KUKA KRL data list: CNC5.dat

&ACCESS RV
DEFDAT CNC5 Public
DECL GLOBAL FRAME gfCNCPoint5[30000]


gfCNCPoint5[1] = {X 169.9145, Y 15.4818, Z -6.3333, A 0.000, B 0.000, C 0.000 }
gfCNCPoint5[2] = {X 169.6699, Y 14.6462, Z -6.3333, A 0.000, B 0.000, C 0.000 }
gfCNCPoint5[3] = {X 169.6011, Y 13.7783, Z -6.3333, A 0.000, B 0.000, C 0.000 }
gfCNCPoint5[4] = {X 169.7111, Y 12.9146, Z -6.3333, A 0.000, B 0.000, C 0.000 }
gfCNCPoint5[5] = {X 169.9952, Y 12.0915, Z -6.3333, A 0.000, B 0.000, C 0.000 }
gfCNCPoint5[6] = {X 170.4414, Y 11.3439, Z -6.3333, A 0.000, B 0.000, C 0.000 }
gfCNCPoint5[7] = {X 171.0309, Y 10.7031, Z -6.3333, A 0.000, B 0.000, C 0.000 }
gfCNCPoint5[8] = {X 171.7389, Y 10.1963, Z -6.3333, A 0.000, B 0.000, C 0.000 }
gfCNCPoint5[9] = {X 172.3689, Y 9.8371, Z -6.3333, A 0.000, B 0.000, C 0.000 }
gfCNCPoint5[10] = {X 173.2226, Y 9.4761, Z -6.3333, A 0.000, B 0.000, C 0.000 }
gfCNCPoint5[11] = {X 174.1343, Y 9.3093, Z -6.3333, A 0.000, B 0.000, C 0.000 }
gfCNCPoint5[12] = {X 175.0605, Y 9.3446, Z -6.3333, A 0.000, B 0.000, C 0.000 }
gfCNCPoint5[13] = {X 175.9569, Y 9.5802, Z -6.3333, A 0.000, B 0.000, C 0.000 }
gfCNCPoint5[14] = {X 177.1785, Y 9.1095, Z -6.3333, A 0.000, B 0.000, C 0.000 }
gfCNCPoint5[15] = {X 179.3486, Y 8.3113, Z -6.3333, A 0.000, B 0.000, C 0.000 }
gfCNCPoint5[16] = {X 181.5872, Y 7.7326, Z -6.3333, A 0.000, B 0.000, C 0.000 }
gfCNCPoint5[17] = {X 183.8722, Y 7.3791, Z -6.3333, A 0.000, B 0.000, C 0.000 }
gfCNCPoint5[18] = {X 186.1811, Y 7.2543, Z -6.3333, A 0.000, B 0.000, C 0.000 }
gfCNCPoint5[19] = {X 188.4909, Y 7.3595, Z -6.3333, A 0.000, B 0.000, C 0.000 }
gfCNCPoint5[20] = {X 190.7789, Y 7.6937, Z -6.3333, A 0.000, B 0.000, C 0.000 }
gfCNCPoint5[21] = {X 192.7312, Y 8.2006, Z -6.3333, A 0.000, B 0.000, C 0.000 }
gfCNCPoint5[22] = {X 194.6099, Y 8.9351, Z -6.3333, A 0.000, B 0.000, C 0.000 }
gfCNCPoint5[23] = {X 196.3884, Y 9.8866, Z -6.3333, A 0.000, B 0.000, C 0.000 }
gfCNCPoint5[24] = {X 198.0419, Y 11.0420, Z -6.3333, A 0.000, B 0.000, C 0.000 }
gfCNCPoint5[25] = {X 199.0952, Y 11.9790, Z -6.3333, A 0.000, B 0.000, C 0.000 }
gfCNCPoint5[26] = {X 200.0403, Y 13.0251, Z -6.3333, A 0.000, B 0.000, C 0.000 }
gfCNCPoint5[27] = {X 200.8660, Y 14.1678, Z -6.3333, A 0.000, B 0.000, C 0.000 }
gfCNCPoint5[28] = {X 201.5625, Y 15.3935, Z -6.3333, A 0.000, B 0.000, C 0.000 }
gfCNCPoint5[29] = {X 202.1217, Y 16.6876, Z -6.3333, A 0.000, B 0.000, C 0.000 }
gfCNCPoint5[30] = {X 202.5931, Y 18.3350, Z -6.3333, A 0.000, B 0.000, C 0.000 }
gfCNCPoint5[31] = {X 202.8729, Y 20.0254, Z -6.3333, A 0.000, B 0.000, C 0.000 }
gfCNCPoint5[32] = {X 202.9574, Y 21.7368, Z -6.3333, A 0.000, B 0.000, C 0.000 }
gfCNCPoint5[33] = {X 202.8453, Y 23.4466, Z -6.3333, A 0.000, B 0.000, C 0.000 }
gfCNCPoint5[34] = {X 202.5383, Y 25.1324, Z -6.3333, A 0.000, B 0.000, C 0.000 }
gfCNCPoint5[35] = {X 202.0887, Y 26.5970, Z -6.3333, A 0.000, B 0.000, C 0.000 }
gfCNCPoint5[36] = {X 201.4503, Y 27.9897, Z -6.3333, A 0.000, B 0.000, C 0.000 }
gfCNCPoint5[37] = {X 200.6341, Y 29.2863, Z -6.3333, A 0.000, B 0.000, C 0.000 }
gfCNCPoint5[38] = {X 199.6544, Y 30.4641, Z -6.3333, A 0.000, B 0.000, C 0.000 }
gfCNCPoint5[39] = {X 198.5281, Y 31.5028, Z -6.3333, A 0.000, B 0.000, C 0.000 }
gfCNCPoint5[40] = {X 199.3593, Y 31.8268, Z -6.3333, A 0.000, B 0.000, C 0.000 }
gfCNCPoint5[41] = {X 200.1043, Y 32.3175, Z -6.3333, A 0.000, B 0.000, C 0.000 }
gfCNCPoint5[42] = {X 200.7302, Y 32.9532, Z -6.3333, A 0.000, B 0.000, C 0.000 }
gfCNCPoint5[43] = {X 201.2091, Y 33.7058, Z -6.3333, A 0.000, B 0.000, C 0.000 }
gfCNCPoint5[44] = {X 204.2502, Y 39.9879, Z -6.3333, A 0.000, B 0.000, C 0.000 }
gfCNCPoint5[45] = {X 204.5648, Y 40.8802, Z -6.3333, A 0.000, B 0.000, C 0.000 }
gfCNCPoint5[46] = {X 204.6737, Y 41.8200, Z -6.3333, A 0.000, B 0.000, C 0.000 }
gfCNCPoint5[47] = {X 204.5715, Y 42.7606, Z -6.3333, A 0.000, B 0.000, C 0.000 }
gfCNCPoint5[48] = {X 204.2633, Y 43.6551, Z -6.3333, A 0.000, B 0.000, C 0.000 }
gfCNCPoint5[49] = {X 203.7643, Y 44.4590, Z -6.3333, A 0.000, B 0.000, C 0.000 }
gfCNCPoint5[50] = {X 203.0996, Y 45.1323, Z -6.3333, A 0.000, B 0.000, C 0.000 }
gfCNCPoint5[51] = {X 202.5635, Y 45.5657, Z -6.3333, A 0.000, B 0.000, C 0.000 }
gfCNCPoint5[52] = {X 201.8660, Y 46.0245, Z -6.3333, A 0.000, B 0.000, C 0.000 }
gfCNCPoint5[53] = {X 201.0922, Y 46.3381, Z -6.3333, A 0.000, B 0.000, C 0.000 }
gfCNCPoint5[54] = {X 200.2721, Y 46.4943, Z -6.3333, A 0.000, B 0.000, C 0.000 }
gfCNCPoint5[55] = {X 199.4373, Y 46.4873, Z -6.3333, A 0.000, B 0.000, C 0.000 }
gfCNCPoint5[56] = {X 198.6199, Y 46.3171, Z -6.3333, A 0.000, B 0.000, C 0.000 }
gfCNCPoint5[57] = {X 196.5061, Y 47.4225, Z -6.3333, A 0.000, B 0.000, C 0.000 }
gfCNCPoint5[58] = {X 194.3068, Y 48.3461, Z -6.3333, A 0.000, B 0.000, C 0.000 }
gfCNCPoint5[59] = {X 192.0377, Y 49.0815, Z -6.3333, A 0.000, B 0.000, C 0.000 }
gfCNCPoint5[60] = {X 189.8324, Y 49.5923, Z -6.3333, A 0.000, B 0.000, C 0.000 }
gfCNCPoint5[61] = {X 187.5867, Y 49.8772, Z -6.3333, A 0.000, B 0.000, C 0.000 }
gfCNCPoint5[62] = {X 185.3237, Y 49.9332, Z -6.3333, A 0.000, B 0.000, C 0.000 }
gfCNCPoint5[63] = {X 183.0667, Y 49.7599, Z -6.3333, A 0.000, B 0.000, C 0.000 }
gfCNCPoint5[64] = {X 180.8388, Y 49.3589, Z -6.3333, A 0.000, B 0.000, C 0.000 }
gfCNCPoint5[65] = {X 179.0075, Y 48.8281, Z -6.3333, A 0.000, B 0.000, C 0.000 }
gfCNCPoint5[66] = {X 177.2496, Y 48.0897, Z -6.3333, A 0.000, B 0.000, C 0.000 }
gfCNCPoint5[67] = {X 175.5885, Y 47.1536, Z -6.3333, A 0.000, B 0.000, C 0.000 }
gfCNCPoint5[68] = {X 174.0464, Y 46.0322, Z -6.3333, A 0.000, B 0.000, C 0.000 }
gfCNCPoint5[69] = {X 172.9127, Y 44.9979, Z -6.3333, A 0.000, B 0.000, C 0.000 }
gfCNCPoint5[70] = {X 171.9093, Y 43.8366, Z -6.3333, A 0.000, B 0.000, C 0.000 }
gfCNCPoint5[71] = {X 171.0504, Y 42.5648, Z -6.3333, A 0.000, B 0.000, C 0.000 }
gfCNCPoint5[72] = {X 170.3480, Y 41.2003, Z -6.3333, A 0.000, B 0.000, C 0.000 }
gfCNCPoint5[73] = {X 169.8121, Y 39.7622, Z -6.3333, A 0.000, B 0.000, C 0.000 }
gfCNCPoint5[74] = {X 169.4500, Y 38.2708, Z -6.3333, A 0.000, B 0.000, C 0.000 }
gfCNCPoint5[75] = {X 169.3946, Y 37.9230, Z -6.3333, A 0.000, B 0.000, C 0.000 }
gfCNCPoint5[76] = {X 165.4444, Y 38.5519, Z -6.3333, A 0.000, B 0.000, C 0.000 }
gfCNCPoint5[77] = {X 165.4444, Y 38.5520, Z -6.3333, A 0.000, B 0.000, C 0.000 }
gfCNCPoint5[78] = {X 169.4737, Y 37.9104, Z -6.3333, A 0.000, B 0.000, C 0.000 }
gfCNCPoint5[79] = {X 169.4183, Y 37.5626, Z -6.3333, A 0.000, B 0.000, C 0.000 }
gfCNCPoint5[80] = {X 169.2618, Y 35.9753, Z -6.3333, A 0.000, B 0.000, C 0.000 }
gfCNCPoint5[81] = {X 169.2787, Y 34.3803, Z -6.3333, A 0.000, B 0.000, C 0.000 }
gfCNCPoint5[82] = {X 169.4688, Y 32.7966, Z -6.3333, A 0.000, B 0.000, C 0.000 }
gfCNCPoint5[83] = {X 169.8298, Y 31.2430, Z -6.3333, A 0.000, B 0.000, C 0.000 }
gfCNCPoint5[84] = {X 170.3575, Y 29.7378, Z -6.3333, A 0.000, B 0.000, C 0.000 }
gfCNCPoint5[85] = {X 171.0238, Y 28.3859, Z -6.3333, A 0.000, B 0.000, C 0.000 }
gfCNCPoint5[86] = {X 171.8736, Y 27.1412, Z -6.3333, A 0.000, B 0.000, C 0.000 }
gfCNCPoint5[87] = {X 172.8900, Y 26.0283, Z -6.3333, A 0.000, B 0.000, C 0.000 }
gfCNCPoint5[88] = {X 174.0526, Y 25.0692, Z -6.3333, A 0.000, B 0.000, C 0.000 }
gfCNCPoint5[89] = {X 175.3386, Y 24.2832, Z -6.3333, A 0.000, B 0.000, C 0.000 }
gfCNCPoint5[90] = {X 174.4745, Y 23.9351, Z -6.3333, A 0.000, B 0.000, C 0.000 }
gfCNCPoint5[91] = {X 173.7095, Y 23.4034, Z -6.3333, A 0.000, B 0.000, C 0.000 }
gfCNCPoint5[92] = {X 173.0820, Y 22.7148, Z -6.3333, A 0.000, B 0.000, C 0.000 }
gfCNCPoint5[93] = {X 172.6235, Y 21.9039, Z -6.3333, A 0.000, B 0.000, C 0.000 }
gfCNCPoint5[94] = {X 169.9886, Y 15.4516, Z -6.3333, A 0.000, B 0.000, C 0.000 }
gfCNCPoint5[95] = {X 169.7252, Y 14.4911, Z -6.3333, A 0.000, B 0.000, C 0.000 }
gfCNCPoint5[96] = {X 169.6977, Y 13.4955, Z -6.3333, A 0.000, B 0.000, C 0.000 }
gfCNCPoint5[97] = {X 169.9076, Y 12.5218, Z -6.3333, A 0.000, B 0.000, C 0.000 }
gfCNCPoint5[98] = {X 170.3429, Y 11.6260, Z -6.3333, A 0.000, B 0.000, C 0.000 }
gfCNCPoint5[99] = {X 170.9787, Y 10.8594, Z -6.3333, A 0.000, B 0.000, C 0.000 }
gfCNCPoint5[100] = {X 171.7785, Y 10.2658, Z -6.3333, A 0.000, B 0.000, C 0.000 }
gfCNCPoint5[101] = {X 172.4082, Y 9.9068, Z -6.3333, A 0.000, B 0.000, C 0.000 }
gfCNCPoint5[102] = {X 173.2457, Y 9.5527, Z -6.3333, A 0.000, B 0.000, C 0.000 }
gfCNCPoint5[103] = {X 174.1402, Y 9.3891, Z -6.3333, A 0.000, B 0.000, C 0.000 }
gfCNCPoint5[104] = {X 175.0488, Y 9.4237, Z -6.3333, A 0.000, B 0.000, C 0.000 }
gfCNCPoint5[105] = {X 175.9283, Y 9.6549, Z -6.3333, A 0.000, B 0.000, C 0.000 }
gfCNCPoint5[106] = {X 176.0174, Y 9.6904, Z -6.3333, A 0.000, B 0.000, C 0.000 }
gfCNCPoint5[107] = {X 177.2098, Y 9.1831, Z -6.3333, A 0.000, B 0.000, C 0.000 }
gfCNCPoint5[108] = {X 179.3724, Y 8.3877, Z -6.3333, A 0.000, B 0.000, C 0.000 }
gfCNCPoint5[109] = {X 181.6033, Y 7.8109, Z -6.3333, A 0.000, B 0.000, C 0.000 }
gfCNCPoint5[110] = {X 183.8805, Y 7.4587, Z -6.3333, A 0.000, B 0.000, C 0.000 }
gfCNCPoint5[111] = {X 186.1814, Y 7.3343, Z -6.3333, A 0.000, B 0.000, C 0.000 }
gfCNCPoint5[112] = {X 188.4833, Y 7.4392, Z -6.3333, A 0.000, B 0.000, C 0.000 }
gfCNCPoint5[113] = {X 190.7634, Y 7.7722, Z -6.3333, A 0.000, B 0.000, C 0.000 }
gfCNCPoint5[114] = {X 192.7066, Y 8.2767, Z -6.3333, A 0.000, B 0.000, C 0.000 }
gfCNCPoint5[115] = {X 194.5764, Y 9.0077, Z -6.3333, A 0.000, B 0.000, C 0.000 }
gfCNCPoint5[116] = {X 196.3466, Y 9.9548, Z -6.3333, A 0.000, B 0.000, C 0.000 }
gfCNCPoint5[117] = {X 197.9923, Y 11.1047, Z -6.3333, A 0.000, B 0.000, C 0.000 }
gfCNCPoint5[118] = {X 199.2842, Y 12.2861, Z -6.3333, A 0.000, B 0.000, C 0.000 }
gfCNCPoint5[119] = {X 200.4037, Y 13.6319, Z -6.3333, A 0.000, B 0.000, C 0.000 }
gfCNCPoint5[120] = {X 201.3302, Y 15.1173, Z -6.3333, A 0.000, B 0.000, C 0.000 }
gfCNCPoint5[121] = {X 202.0464, Y 16.7147, Z -6.3333, A 0.000, B 0.000, C 0.000 }
gfCNCPoint5[122] = {X 202.5152, Y 18.3531, Z -6.3333, A 0.000, B 0.000, C 0.000 }
gfCNCPoint5[123] = {X 202.7934, Y 20.0344, Z -6.3333, A 0.000, B 0.000, C 0.000 }
gfCNCPoint5[124] = {X 202.8774, Y 21.7366, Z -6.3333, A 0.000, B 0.000, C 0.000 }
gfCNCPoint5[125] = {X 202.7659, Y 23.4371, Z -6.3333, A 0.000, B 0.000, C 0.000 }
gfCNCPoint5[126] = {X 202.4605, Y 25.1137, Z -6.3333, A 0.000, B 0.000, C 0.000 }
gfCNCPoint5[127] = {X 202.0025, Y 26.5984, Z -6.3333, A 0.000, B 0.000, C 0.000 }
gfCNCPoint5[128] = {X 201.3492, Y 28.0081, Z -6.3333, A 0.000, B 0.000, C 0.000 }
gfCNCPoint5[129] = {X 200.5123, Y 29.3172, Z -6.3333, A 0.000, B 0.000, C 0.000 }
gfCNCPoint5[130] = {X 199.5071, Y 30.5019, Z -6.3333, A 0.000, B 0.000, C 0.000 }
gfCNCPoint5[131] = {X 198.3518, Y 31.5408, Z -6.3333, A 0.000, B 0.000, C 0.000 }
gfCNCPoint5[132] = {X 199.2151, Y 31.8442, Z -6.3333, A 0.000, B 0.000, C 0.000 }
gfCNCPoint5[133] = {X 199.9912, Y 32.3290, Z -6.3333, A 0.000, B 0.000, C 0.000 }
gfCNCPoint5[134] = {X 200.6425, Y 32.9718, Z -6.3333, A 0.000, B 0.000, C 0.000 }
gfCNCPoint5[135] = {X 201.1375, Y 33.7414, Z -6.3333, A 0.000, B 0.000, C 0.000 }
gfCNCPoint5[136] = {X 204.1781, Y 40.0227, Z -6.3333, A 0.000, B 0.000, C 0.000 }
gfCNCPoint5[137] = {X 204.4868, Y 40.8982, Z -6.3333, A 0.000, B 0.000, C 0.000 }
gfCNCPoint5[138] = {X 204.5937, Y 41.8203, Z -6.3333, A 0.000, B 0.000, C 0.000 }
gfCNCPoint5[139] = {X 204.4934, Y 42.7431, Z -6.3333, A 0.000, B 0.000, C 0.000 }
gfCNCPoint5[140] = {X 204.1910, Y 43.6208, Z -6.3333, A 0.000, B 0.000, C 0.000 }
gfCNCPoint5[141] = {X 203.7015, Y 44.4095, Z -6.3333, A 0.000, B 0.000, C 0.000 }
gfCNCPoint5[142] = {X 203.0493, Y 45.0700, Z -6.3333, A 0.000, B 0.000, C 0.000 }
gfCNCPoint5[143] = {X 202.5132, Y 45.5035, Z -6.3333, A 0.000, B 0.000, C 0.000 }
gfCNCPoint5[144] = {X 201.8226, Y 45.9569, Z -6.3333, A 0.000, B 0.000, C 0.000 }
gfCNCPoint5[145] = {X 201.0562, Y 46.2653, Z -6.3333, A 0.000, B 0.000, C 0.000 }
gfCNCPoint5[146] = {X 200.2440, Y 46.4165, Z -6.3333, A 0.000, B 0.000, C 0.000 }
gfCNCPoint5[147] = {X 199.4179, Y 46.4046, Z -6.3333, A 0.000, B 0.000, C 0.000 }
gfCNCPoint5[148] = {X 198.6104, Y 46.2302, Z -6.3333, A 0.000, B 0.000, C 0.000 }
gfCNCPoint5[149] = {X 196.4932, Y 47.3401, Z -6.3333, A 0.000, B 0.000, C 0.000 }
gfCNCPoint5[150] = {X 194.2898, Y 48.2671, Z -6.3333, A 0.000, B 0.000, C 0.000 }
gfCNCPoint5[151] = {X 192.0159, Y 49.0046, Z -6.3333, A 0.000, B 0.000, C 0.000 }
gfCNCPoint5[152] = {X 189.8184, Y 49.5135, Z -6.3333, A 0.000, B 0.000, C 0.000 }
gfCNCPoint5[153] = {X 187.5807, Y 49.7974, Z -6.3333, A 0.000, B 0.000, C 0.000 }
gfCNCPoint5[154] = {X 185.3258, Y 49.8532, Z -6.3333, A 0.000, B 0.000, C 0.000 }
gfCNCPoint5[155] = {X 183.0767, Y 49.6805, Z -6.3333, A 0.000, B 0.000, C 0.000 }
gfCNCPoint5[156] = {X 180.8568, Y 49.2809, Z -6.3333, A 0.000, B 0.000, C 0.000 }
gfCNCPoint5[157] = {X 179.0342, Y 48.7527, Z -6.3333, A 0.000, B 0.000, C 0.000 }
gfCNCPoint5[158] = {X 177.2847, Y 48.0178, Z -6.3333, A 0.000, B 0.000, C 0.000 }
gfCNCPoint5[159] = {X 175.6316, Y 47.0862, Z -6.3333, A 0.000, B 0.000, C 0.000 }
gfCNCPoint5[160] = {X 174.0969, Y 45.9702, Z -6.3333, A 0.000, B 0.000, C 0.000 }
gfCNCPoint5[161] = {X 172.9702, Y 44.9423, Z -6.3333, A 0.000, B 0.000, C 0.000 }
gfCNCPoint5[162] = {X 171.9731, Y 43.7883, Z -6.3333, A 0.000, B 0.000, C 0.000 }
gfCNCPoint5[163] = {X 171.1195, Y 42.5245, Z -6.3333, A 0.000, B 0.000, C 0.000 }
gfCNCPoint5[164] = {X 170.4215, Y 41.1685, Z -6.3333, A 0.000, B 0.000, C 0.000 }
gfCNCPoint5[165] = {X 169.8888, Y 39.7395, Z -6.3333, A 0.000, B 0.000, C 0.000 }
gfCNCPoint5[166] = {X 169.5289, Y 38.2574, Z -6.3333, A 0.000, B 0.000, C 0.000 }
gfCNCPoint5[167] = {X 169.4737, Y 37.9104, Z -6.3333, A 0.000, B 0.000, C 0.000 }
gfCNCPoint5[168] = {X 165.5234, Y 38.5394, Z -6.3333, A 0.000, B 0.000, C 0.000 }
gfCNCPoint5[169] = {X 169.5527, Y 37.8979, Z -6.3333, A 0.000, B 0.000, C 0.000 }
gfCNCPoint5[170] = {X 169.4973, Y 37.5504, Z -6.3333, A 0.000, B 0.000, C 0.000 }
gfCNCPoint5[171] = {X 169.3417, Y 35.9717, Z -6.3333, A 0.000, B 0.000, C 0.000 }
gfCNCPoint5[172] = {X 169.3585, Y 34.3854, Z -6.3333, A 0.000, B 0.000, C 0.000 }
gfCNCPoint5[173] = {X 169.5476, Y 32.8104, Z -6.3333, A 0.000, B 0.000, C 0.000 }
gfCNCPoint5[174] = {X 169.9067, Y 31.2652, Z -6.3333, A 0.000, B 0.000, C 0.000 }
gfCNCPoint5[175] = {X 170.4315, Y 29.7681, Z -6.3333, A 0.000, B 0.000, C 0.000 }
gfCNCPoint5[176] = {X 171.1145, Y 28.3894, Z -6.3333, A 0.000, B 0.000, C 0.000 }
gfCNCPoint5[177] = {X 171.9897, Y 27.1240, Z -6.3333, A 0.000, B 0.000, C 0.000 }
gfCNCPoint5[178] = {X 173.0386, Y 25.9983, Z -6.3333, A 0.000, B 0.000, C 0.000 }
gfCNCPoint5[179] = {X 174.2393, Y 25.0361, Z -6.3333, A 0.000, B 0.000, C 0.000 }
gfCNCPoint5[180] = {X 175.5664, Y 24.2576, Z -6.3333, A 0.000, B 0.000, C 0.000 }
gfCNCPoint5[181] = {X 174.6545, Y 23.9378, Z -6.3333, A 0.000, B 0.000, C 0.000 }
gfCNCPoint5[182] = {X 173.8434, Y 23.4125, Z -6.3333, A 0.000, B 0.000, C 0.000 }
gfCNCPoint5[183] = {X 173.1785, Y 22.7111, Z -6.3333, A 0.000, B 0.000, C 0.000 }
gfCNCPoint5[184] = {X 172.6973, Y 21.8731, Z -6.3333, A 0.000, B 0.000, C 0.000 }
gfCNCPoint5[185] = {X 170.0626, Y 15.4213, Z -6.3333, A 0.000, B 0.000, C 0.000 }
gfCNCPoint5[186] = {X 169.8043, Y 14.4793, Z -6.3333, A 0.000, B 0.000, C 0.000 }
gfCNCPoint5[187] = {X 169.7773, Y 13.5028, Z -6.3333, A 0.000, B 0.000, C 0.000 }
gfCNCPoint5[188] = {X 169.9832, Y 12.5479, Z -6.3333, A 0.000, B 0.000, C 0.000 }
gfCNCPoint5[189] = {X 170.4102, Y 11.6694, Z -6.3333, A 0.000, B 0.000, C 0.000 }
gfCNCPoint5[190] = {X 171.0337, Y 10.9174, Z -6.3333, A 0.000, B 0.000, C 0.000 }
gfCNCPoint5[191] = {X 171.8181, Y 10.3353, Z -6.3333, A 0.000, B 0.000, C 0.000 }
gfCNCPoint5[192] = {X 172.4475, Y 9.9764, Z -6.3333, A 0.000, B 0.000, C 0.000 }
gfCNCPoint5[193] = {X 173.2689, Y 9.6293, Z -6.3333, A 0.000, B 0.000, C 0.000 }
gfCNCPoint5[194] = {X 174.1461, Y 9.4689, Z -6.3333, A 0.000, B 0.000, C 0.000 }
gfCNCPoint5[195] = {X 175.0372, Y 9.5028, Z -6.3333, A 0.000, B 0.000, C 0.000 }
gfCNCPoint5[196] = {X 175.8996, Y 9.7296, Z -6.3333, A 0.000, B 0.000, C 0.000 }
gfCNCPoint5[197] = {X 175.9650, Y 9.7554, Z -6.3333, A 0.000, B 0.000, C 0.000 }
gfCNCPoint5[198] = {X 176.0299, Y 9.7822, Z -6.3333, A 0.000, B 0.000, C 0.000 }
gfCNCPoint5[199] = {X 176.0576, Y 9.7602, Z -6.3333, A 0.000, B 0.000, C 0.000 }
gfCNCPoint5[200] = {X 177.2411, Y 9.2567, Z -6.3333, A 0.000, B 0.000, C 0.000 }
gfCNCPoint5[201] = {X 179.3963, Y 8.4640, Z -6.3333, A 0.000, B 0.000, C 0.000 }
gfCNCPoint5[202] = {X 181.6195, Y 7.8893, Z -6.3333, A 0.000, B 0.000, C 0.000 }
gfCNCPoint5[203] = {X 183.8888, Y 7.5382, Z -6.3333, A 0.000, B 0.000, C 0.000 }
gfCNCPoint5[204] = {X 186.1818, Y 7.4143, Z -6.3333, A 0.000, B 0.000, C 0.000 }
gfCNCPoint5[205] = {X 188.4757, Y 7.5188, Z -6.3333, A 0.000, B 0.000, C 0.000 }
gfCNCPoint5[206] = {X 190.7479, Y 7.8506, Z -6.3333, A 0.000, B 0.000, C 0.000 }
gfCNCPoint5[207] = {X 192.6819, Y 8.3528, Z -6.3333, A 0.000, B 0.000, C 0.000 }
gfCNCPoint5[208] = {X 194.5429, Y 9.0804, Z -6.3333, A 0.000, B 0.000, C 0.000 }
gfCNCPoint5[209] = {X 196.3047, Y 10.0230, Z -6.3333, A 0.000, B 0.000, C 0.000 }
gfCNCPoint5[210] = {X 197.9426, Y 11.1675, Z -6.3333, A 0.000, B 0.000, C 0.000 }
gfCNCPoint5[211] = {X 199.2263, Y 12.3413, Z -6.3333, A 0.000, B 0.000, C 0.000 }
gfCNCPoint5[212] = {X 200.3388, Y 13.6786, Z -6.3333, A 0.000, B 0.000, C 0.000 }
gfCNCPoint5[213] = {X 201.2594, Y 15.1545, Z -6.3333, A 0.000, B 0.000, C 0.000 }
gfCNCPoint5[214] = {X 201.9711, Y 16.7417, Z -6.3333, A 0.000, B 0.000, C 0.000 }
gfCNCPoint5[215] = {X 202.4373, Y 18.3713, Z -6.3333, A 0.000, B 0.000, C 0.000 }
gfCNCPoint5[216] = {X 202.7139, Y 20.0435, Z -6.3333, A 0.000, B 0.000, C 0.000 }
gfCNCPoint5[217] = {X 202.7974, Y 21.7363, Z -6.3333, A 0.000, B 0.000, C 0.000 }
gfCNCPoint5[218] = {X 202.6865, Y 23.4276, Z -6.3333, A 0.000, B 0.000, C 0.000 }
gfCNCPoint5[219] = {X 202.3827, Y 25.0951, Z -6.3333, A 0.000, B 0.000, C 0.000 }
gfCNCPoint5[220] = {X 201.9155, Y 26.6018, Z -6.3333, A 0.000, B 0.000, C 0.000 }
gfCNCPoint5[221] = {X 201.2457, Y 28.0301, Z -6.3333, A 0.000, B 0.000, C 0.000 }
gfCNCPoint5[222] = {X 200.3860, Y 29.3527, Z -6.3333, A 0.000, B 0.000, C 0.000 }
gfCNCPoint5[223] = {X 199.3528, Y 30.5447, Z -6.3333, A 0.000, B 0.000, C 0.000 }
gfCNCPoint5[224] = {X 198.1656, Y 31.5835, Z -6.3333, A 0.000, B 0.000, C 0.000 }
gfCNCPoint5[225] = {X 199.0634, Y 31.8623, Z -6.3333, A 0.000, B 0.000, C 0.000 }
gfCNCPoint5[226] = {X 199.8735, Y 32.3392, Z -6.3333, A 0.000, B 0.000, C 0.000 }
gfCNCPoint5[227] = {X 200.5529, Y 32.9888, Z -6.3333, A 0.000, B 0.000, C 0.000 }
gfCNCPoint5[228] = {X 201.0657, Y 33.7766, Z -6.3333, A 0.000, B 0.000, C 0.000 }
gfCNCPoint5[229] = {X 204.1061, Y 40.0576, Z -6.3333, A 0.000, B 0.000, C 0.000 }
gfCNCPoint5[230] = {X 204.4089, Y 40.9162, Z -6.3333, A 0.000, B 0.000, C 0.000 }
gfCNCPoint5[231] = {X 204.5137, Y 41.8206, Z -6.3333, A 0.000, B 0.000, C 0.000 }
gfCNCPoint5[232] = {X 204.4154, Y 42.7257, Z -6.3333, A 0.000, B 0.000, C 0.000 }
gfCNCPoint5[233] = {X 204.1188, Y 43.5864, Z -6.3333, A 0.000, B 0.000, C 0.000 }
gfCNCPoint5[234] = {X 203.6387, Y 44.3600, Z -6.3333, A 0.000, B 0.000, C 0.000 }
gfCNCPoint5[235] = {X 202.9990, Y 45.0078, Z -6.3333, A 0.000, B 0.000, C 0.000 }
gfCNCPoint5[236] = {X 202.4629, Y 45.4413, Z -6.3333, A 0.000, B 0.000, C 0.000 }
gfCNCPoint5[237] = {X 201.7792, Y 45.8893, Z -6.3333, A 0.000, B 0.000, C 0.000 }
gfCNCPoint5[238] = {X 201.0202, Y 46.1924, Z -6.3333, A 0.000, B 0.000, C 0.000 }
gfCNCPoint5[239] = {X 200.2160, Y 46.3385, Z -6.3333, A 0.000, B 0.000, C 0.000 }
gfCNCPoint5[240] = {X 199.3988, Y 46.3218, Z -6.3333, A 0.000, B 0.000, C 0.000 }
gfCNCPoint5[241] = {X 198.6013, Y 46.1430, Z -6.3333, A 0.000, B 0.000, C 0.000 }
gfCNCPoint5[242] = {X 196.4806, Y 47.2576, Z -6.3333, A 0.000, B 0.000, C 0.000 }
gfCNCPoint5[243] = {X 194.2730, Y 48.1880, Z -6.3333, A 0.000, B 0.000, C 0.000 }
gfCNCPoint5[244] = {X 191.9942, Y 48.9276, Z -6.3333, A 0.000, B 0.000, C 0.000 }
gfCNCPoint5[245] = {X 189.8046, Y 49.4347, Z -6.3333, A 0.000, B 0.000, C 0.000 }
gfCNCPoint5[246] = {X 187.5748, Y 49.7176, Z -6.3333, A 0.000, B 0.000, C 0.000 }
gfCNCPoint5[247] = {X 185.3279, Y 49.7733, Z -6.3333, A 0.000, B 0.000, C 0.000 }
gfCNCPoint5[248] = {X 183.0868, Y 49.6011, Z -6.3333, A 0.000, B 0.000, C 0.000 }
gfCNCPoint5[249] = {X 180.8747, Y 49.2030, Z -6.3333, A 0.000, B 0.000, C 0.000 }
gfCNCPoint5[250] = {X 179.0610, Y 48.6773, Z -6.3333, A 0.000, B 0.000, C 0.000 }
gfCNCPoint5[251] = {X 177.3199, Y 47.9460, Z -6.3333, A 0.000, B 0.000, C 0.000 }
gfCNCPoint5[252] = {X 175.6747, Y 47.0188, Z -6.3333, A 0.000, B 0.000, C 0.000 }
gfCNCPoint5[253] = {X 174.1474, Y 45.9081, Z -6.3333, A 0.000, B 0.000, C 0.000 }
gfCNCPoint5[254] = {X 173.0278, Y 44.8867, Z -6.3333, A 0.000, B 0.000, C 0.000 }
gfCNCPoint5[255] = {X 172.0369, Y 43.7400, Z -6.3333, A 0.000, B 0.000, C 0.000 }
gfCNCPoint5[256] = {X 171.1886, Y 42.4842, Z -6.3333, A 0.000, B 0.000, C 0.000 }
gfCNCPoint5[257] = {X 170.4949, Y 41.1367, Z -6.3333, A 0.000, B 0.000, C 0.000 }
gfCNCPoint5[258] = {X 169.9655, Y 39.7167, Z -6.3333, A 0.000, B 0.000, C 0.000 }
gfCNCPoint5[259] = {X 169.6078, Y 38.2440, Z -6.3333, A 0.000, B 0.000, C 0.000 }
gfCNCPoint5[260] = {X 169.5527, Y 37.8979, Z -6.3333, A 0.000, B 0.000, C 0.000 }
gfCNCPoint5[261] = {X 165.6024, Y 38.5268, Z -6.3333, A 0.000, B 0.000, C 0.000 }
gfCNCPoint5[262] = {X 169.6317, Y 37.8853, Z -6.3333, A 0.000, B 0.000, C 0.000 }
gfCNCPoint5[263] = {X 169.5764, Y 37.5383, Z -6.3333, A 0.000, B 0.000, C 0.000 }
gfCNCPoint5[264] = {X 169.4216, Y 35.9682, Z -6.3333, A 0.000, B 0.000, C 0.000 }
gfCNCPoint5[265] = {X 169.4384, Y 34.3906, Z -6.3333, A 0.000, B 0.000, C 0.000 }
gfCNCPoint5[266] = {X 169.6264, Y 32.8241, Z -6.3333, A 0.000, B 0.000, C 0.000 }
gfCNCPoint5[267] = {X 169.9835, Y 31.2873, Z -6.3333, A 0.000, B 0.000, C 0.000 }
gfCNCPoint5[268] = {X 170.5055, Y 29.7985, Z -6.3333, A 0.000, B 0.000, C 0.000 }
gfCNCPoint5[269] = {X 171.2081, Y 28.3884, Z -6.3333, A 0.000, B 0.000, C 0.000 }
gfCNCPoint5[270] = {X 172.1131, Y 27.0989, Z -6.3333, A 0.000, B 0.000, C 0.000 }
gfCNCPoint5[271] = {X 173.2003, Y 25.9588, Z -6.3333, A 0.000, B 0.000, C 0.000 }
gfCNCPoint5[272] = {X 174.4454, Y 24.9935, Z -6.3333, A 0.000, B 0.000, C 0.000 }
gfCNCPoint5[273] = {X 175.8205, Y 24.2247, Z -6.3333, A 0.000, B 0.000, C 0.000 }
gfCNCPoint5[274] = {X 175.0297, Y 24.0136, Z -6.3333, A 0.000, B 0.000, C 0.000 }
gfCNCPoint5[275] = {X 174.2985, Y 23.6460, Z -6.3333, A 0.000, B 0.000, C 0.000 }
gfCNCPoint5[276] = {X 173.6573, Y 23.1373, Z -6.3333, A 0.000, B 0.000, C 0.000 }
gfCNCPoint5[277] = {X 173.1332, Y 22.5087, Z -6.3333, A 0.000, B 0.000, C 0.000 }
gfCNCPoint5[278] = {X 172.7479, Y 21.7866, Z -6.3333, A 0.000, B 0.000, C 0.000 }
gfCNCPoint5[279] = {X 170.1367, Y 15.3911, Z -6.3333, A 0.000, B 0.000, C 0.000 }
gfCNCPoint5[280] = {X 169.8835, Y 14.4675, Z -6.3333, A 0.000, B 0.000, C 0.000 }
gfCNCPoint5[281] = {X 169.8570, Y 13.5102, Z -6.3333, A 0.000, B 0.000, C 0.000 }
gfCNCPoint5[282] = {X 170.0588, Y 12.5740, Z -6.3333, A 0.000, B 0.000, C 0.000 }
gfCNCPoint5[283] = {X 170.4774, Y 11.7127, Z -6.3333, A 0.000, B 0.000, C 0.000 }
gfCNCPoint5[284] = {X 171.0888, Y 10.9755, Z -6.3333, A 0.000, B 0.000, C 0.000 }
gfCNCPoint5[285] = {X 171.8578, Y 10.4048, Z -6.3333, A 0.000, B 0.000, C 0.000 }
gfCNCPoint5[286] = {X 172.4867, Y 10.0462, Z -6.3333, A 0.000, B 0.000, C 0.000 }
gfCNCPoint5[287] = {X 173.2919, Y 9.7059, Z -6.3333, A 0.000, B 0.000, C 0.000 }
gfCNCPoint5[288] = {X 174.1519, Y 9.5486, Z -6.3333, A 0.000, B 0.000, C 0.000 }
gfCNCPoint5[289] = {X 175.0254, Y 9.5820, Z -6.3333, A 0.000, B 0.000, C 0.000 }
gfCNCPoint5[290] = {X 175.8709, Y 9.8043, Z -6.3333, A 0.000, B 0.000, C 0.000 }
gfCNCPoint5[291] = {X 175.9569, Y 9.8385, Z -6.3333, A 0.000, B 0.000, C 0.000 }
gfCNCPoint5[292] = {X 176.0421, Y 9.8746, Z -6.3333, A 0.000, B 0.000, C 0.000 }
gfCNCPoint5[293] = {X 176.0989, Y 9.8296, Z -6.3333, A 0.000, B 0.000, C 0.000 }
gfCNCPoint5[294] = {X 177.2724, Y 9.3303, Z -6.3333, A 0.000, B 0.000, C 0.000 }
gfCNCPoint5[295] = {X 179.4201, Y 8.5404, Z -6.3333, A 0.000, B 0.000, C 0.000 }
gfCNCPoint5[296] = {X 181.6356, Y 7.9676, Z -6.3333, A 0.000, B 0.000, C 0.000 }
gfCNCPoint5[297] = {X 183.8971, Y 7.6178, Z -6.3333, A 0.000, B 0.000, C 0.000 }
gfCNCPoint5[298] = {X 186.1821, Y 7.4943, Z -6.3333, A 0.000, B 0.000, C 0.000 }
gfCNCPoint5[299] = {X 188.4681, Y 7.5985, Z -6.3333, A 0.000, B 0.000, C 0.000 }
gfCNCPoint5[300] = {X 190.7324, Y 7.9291, Z -6.3333, A 0.000, B 0.000, C 0.000 }
gfCNCPoint5[301] = {X 192.6573, Y 8.4289, Z -6.3333, A 0.000, B 0.000, C 0.000 }
gfCNCPoint5[302] = {X 194.5094, Y 9.1530, Z -6.3333, A 0.000, B 0.000, C 0.000 }
gfCNCPoint5[303] = {X 196.2629, Y 10.0912, Z -6.3333, A 0.000, B 0.000, C 0.000 }
gfCNCPoint5[304] = {X 197.8930, Y 11.2302, Z -6.3333, A 0.000, B 0.000, C 0.000 }
gfCNCPoint5[305] = {X 199.1685, Y 12.3966, Z -6.3333, A 0.000, B 0.000, C 0.000 }
gfCNCPoint5[306] = {X 200.2738, Y 13.7253, Z -6.3333, A 0.000, B 0.000, C 0.000 }
gfCNCPoint5[307] = {X 201.1885, Y 15.1917, Z -6.3333, A 0.000, B 0.000, C 0.000 }
gfCNCPoint5[308] = {X 201.8958, Y 16.7687, Z -6.3333, A 0.000, B 0.000, C 0.000 }
gfCNCPoint5[309] = {X 202.3594, Y 18.3894, Z -6.3333, A 0.000, B 0.000, C 0.000 }
gfCNCPoint5[310] = {X 202.6344, Y 20.0525, Z -6.3333, A 0.000, B 0.000, C 0.000 }
gfCNCPoint5[311] = {X 202.7174, Y 21.7361, Z -6.3333, A 0.000, B 0.000, C 0.000 }
gfCNCPoint5[312] = {X 202.6070, Y 23.4182, Z -6.3333, A 0.000, B 0.000, C 0.000 }
gfCNCPoint5[313] = {X 202.3049, Y 25.0766, Z -6.3333, A 0.000, B 0.000, C 0.000 }
gfCNCPoint5[314] = {X 201.8273, Y 26.6077, Z -6.3333, A 0.000, B 0.000, C 0.000 }
gfCNCPoint5[315] = {X 201.1392, Y 28.0565, Z -6.3333, A 0.000, B 0.000, C 0.000 }
gfCNCPoint5[316] = {X 200.2541, Y 29.3941, Z -6.3333, A 0.000, B 0.000, C 0.000 }
gfCNCPoint5[317] = {X 199.1896, Y 30.5939, Z -6.3333, A 0.000, B 0.000, C 0.000 }
gfCNCPoint5[318] = {X 197.9670, Y 31.6320, Z -6.3333, A 0.000, B 0.000, C 0.000 }
gfCNCPoint5[319] = {X 198.7286, Y 31.8161, Z -6.3333, A 0.000, B 0.000, C 0.000 }
gfCNCPoint5[320] = {X 199.4396, Y 32.1451, Z -6.3333, A 0.000, B 0.000, C 0.000 }
gfCNCPoint5[321] = {X 200.0729, Y 32.6064, Z -6.3333, A 0.000, B 0.000, C 0.000 }
gfCNCPoint5[322] = {X 200.6042, Y 33.1823, Z -6.3333, A 0.000, B 0.000, C 0.000 }
gfCNCPoint5[323] = {X 201.0129, Y 33.8507, Z -6.3333, A 0.000, B 0.000, C 0.000 }
gfCNCPoint5[324] = {X 204.0341, Y 40.0925, Z -6.3333, A 0.000, B 0.000, C 0.000 }
gfCNCPoint5[325] = {X 204.3309, Y 40.9342, Z -6.3333, A 0.000, B 0.000, C 0.000 }
gfCNCPoint5[326] = {X 204.4337, Y 41.8209, Z -6.3333, A 0.000, B 0.000, C 0.000 }
gfCNCPoint5[327] = {X 204.3373, Y 42.7082, Z -6.3333, A 0.000, B 0.000, C 0.000 }
gfCNCPoint5[328] = {X 204.0465, Y 43.5521, Z -6.3333, A 0.000, B 0.000, C 0.000 }
gfCNCPoint5[329] = {X 203.5758, Y 44.3105, Z -6.3333, A 0.000, B 0.000, C 0.000 }
gfCNCPoint5[330] = {X 202.9487, Y 44.9456, Z -6.3333, A 0.000, B 0.000, C 0.000 }
gfCNCPoint5[331] = {X 202.4125, Y 45.3791, Z -6.3333, A 0.000, B 0.000, C 0.000 }
gfCNCPoint5[332] = {X 201.7359, Y 45.8217, Z -6.3333, A 0.000, B 0.000, C 0.000 }
gfCNCPoint5[333] = {X 200.9842, Y 46.1195, Z -6.3333, A 0.000, B 0.000, C 0.000 }
gfCNCPoint5[334] = {X 200.1881, Y 46.2604, Z -6.3333, A 0.000, B 0.000, C 0.000 }
gfCNCPoint5[335] = {X 199.3799, Y 46.2388, Z -6.3333, A 0.000, B 0.000, C 0.000 }
gfCNCPoint5[336] = {X 198.5924, Y 46.0556, Z -6.3333, A 0.000, B 0.000, C 0.000 }
gfCNCPoint5[337] = {X 196.4682, Y 47.1749, Z -6.3333, A 0.000, B 0.000, C 0.000 }
gfCNCPoint5[338] = {X 194.2562, Y 48.1089, Z -6.3333, A 0.000, B 0.000, C 0.000 }
gfCNCPoint5[339] = {X 191.9725, Y 48.8506, Z -6.3333, A 0.000, B 0.000, C 0.000 }
gfCNCPoint5[340] = {X 189.7907, Y 49.3559, Z -6.3333, A 0.000, B 0.000, C 0.000 }
gfCNCPoint5[341] = {X 187.5689, Y 49.6378, Z -6.3333, A 0.000, B 0.000, C 0.000 }
gfCNCPoint5[342] = {X 185.3300, Y 49.6933, Z -6.3333, A 0.000, B 0.000, C 0.000 }
gfCNCPoint5[343] = {X 183.0969, Y 49.5218, Z -6.3333, A 0.000, B 0.000, C 0.000 }
gfCNCPoint5[344] = {X 180.8928, Y 49.1251, Z -6.3333, A 0.000, B 0.000, C 0.000 }
gfCNCPoint5[345] = {X 179.0877, Y 48.6019, Z -6.3333, A 0.000, B 0.000, C 0.000 }
gfCNCPoint5[346] = {X 177.3550, Y 47.8741, Z -6.3333, A 0.000, B 0.000, C 0.000 }
gfCNCPoint5[347] = {X 175.7178, Y 46.9514, Z -6.3333, A 0.000, B 0.000, C 0.000 }
gfCNCPoint5[348] = {X 174.1979, Y 45.8461, Z -6.3333, A 0.000, B 0.000, C 0.000 }
gfCNCPoint5[349] = {X 173.0854, Y 44.8312, Z -6.3333, A 0.000, B 0.000, C 0.000 }
gfCNCPoint5[350] = {X 172.1007, Y 43.6918, Z -6.3333, A 0.000, B 0.000, C 0.000 }
gfCNCPoint5[351] = {X 171.2577, Y 42.4439, Z -6.3333, A 0.000, B 0.000, C 0.000 }
gfCNCPoint5[352] = {X 170.5683, Y 41.1050, Z -6.3333, A 0.000, B 0.000, C 0.000 }
gfCNCPoint5[353] = {X 170.0422, Y 39.6940, Z -6.3333, A 0.000, B 0.000, C 0.000 }
gfCNCPoint5[354] = {X 169.6866, Y 38.2306, Z -6.3333, A 0.000, B 0.000, C 0.000 }
gfCNCPoint5[355] = {X 169.6317, Y 37.8853, Z -6.3333, A 0.000, B 0.000, C 0.000 }
gfCNCPoint5[356] = {X 165.6024, Y 38.5268, Z -6.3333, A 0.000, B 0.000, C 0.000 }
gfCNCPoint5[357] = {X 165.6024, Y 38.5268, Z -3.3333, A 0.000, B 0.000, C 0.000 }
gfCNCPoint5[358] = {X 165.6024, Y 38.5268, Z 11.0000, A 0.000, B 0.000, C 0.000 }
gfCNCPoint5[359] = {X 210.1642, Y 28.5738, Z 11.0000, A 0.000, B 0.000, C 0.000 }
gfCNCPoint5[360] = {X 210.1642, Y 28.5738, Z -3.3333, A 0.000, B 0.000, C 0.000 }
gfCNCPoint5[361] = {X 210.1642, Y 28.5738, Z -6.3333, A 0.000, B 0.000, C 0.000 }
gfCNCPoint5[362] = {X 214.2442, Y 28.5738, Z -6.3333, A 0.000, B 0.000, C 0.000 }
gfCNCPoint5[363] = {X 214.2442, Y 17.4624, Z -6.3333, A 0.000, B 0.000, C 0.000 }
gfCNCPoint5[364] = {X 214.2389, Y 16.7692, Z -6.3333, A 0.000, B 0.000, C 0.000 }
gfCNCPoint5[365] = {X 214.2422, Y 16.2722, Z -6.3333, A 0.000, B 0.000, C 0.000 }
gfCNCPoint5[366] = {X 213.6045, Y 15.6011, Z -6.3333, A 0.000, B 0.000, C 0.000 }
gfCNCPoint5[367] = {X 213.1245, Y 14.8095, Z -6.3333, A 0.000, B 0.000, C 0.000 }
gfCNCPoint5[368] = {X 212.8241, Y 13.9339, Z -6.3333, A 0.000, B 0.000, C 0.000 }
gfCNCPoint5[369] = {X 212.7172, Y 13.0143, Z -6.3333, A 0.000, B 0.000, C 0.000 }
gfCNCPoint5[370] = {X 212.7170, Y 12.1868, Z -6.3333, A 0.000, B 0.000, C 0.000 }
gfCNCPoint5[371] = {X 212.8253, Y 11.2255, Z -6.3333, A 0.000, B 0.000, C 0.000 }
gfCNCPoint5[372] = {X 213.1448, Y 10.3124, Z -6.3333, A 0.000, B 0.000, C 0.000 }
gfCNCPoint5[373] = {X 213.6595, Y 9.4933, Z -6.3333, A 0.000, B 0.000, C 0.000 }
gfCNCPoint5[374] = {X 214.3435, Y 8.8093, Z -6.3333, A 0.000, B 0.000, C 0.000 }
gfCNCPoint5[375] = {X 215.1626, Y 8.2946, Z -6.3333, A 0.000, B 0.000, C 0.000 }
gfCNCPoint5[376] = {X 216.0757, Y 7.9751, Z -6.3333, A 0.000, B 0.000, C 0.000 }
gfCNCPoint5[377] = {X 217.0370, Y 7.8668, Z -6.3333, A 0.000, B 0.000, C 0.000 }
gfCNCPoint5[378] = {X 223.4805, Y 7.8668, Z -6.3333, A 0.000, B 0.000, C 0.000 }
gfCNCPoint5[379] = {X 224.4418, Y 7.9751, Z -6.3333, A 0.000, B 0.000, C 0.000 }
gfCNCPoint5[380] = {X 225.3549, Y 8.2946, Z -6.3333, A 0.000, B 0.000, C 0.000 }
gfCNCPoint5[381] = {X 226.1740, Y 8.8093, Z -6.3333, A 0.000, B 0.000, C 0.000 }
gfCNCPoint5[382] = {X 226.8580, Y 9.4933, Z -6.3333, A 0.000, B 0.000, C 0.000 }
gfCNCPoint5[383] = {X 227.3727, Y 10.3124, Z -6.3333, A 0.000, B 0.000, C 0.000 }
gfCNCPoint5[384] = {X 227.6922, Y 11.2255, Z -6.3333, A 0.000, B 0.000, C 0.000 }
gfCNCPoint5[385] = {X 227.8005, Y 12.1868, Z -6.3333, A 0.000, B 0.000, C 0.000 }
gfCNCPoint5[386] = {X 227.8005, Y 12.9782, Z -6.3333, A 0.000, B 0.000, C 0.000 }
gfCNCPoint5[387] = {X 227.6992, Y 13.9079, Z -6.3333, A 0.000, B 0.000, C 0.000 }
gfCNCPoint5[388] = {X 227.4003, Y 14.7940, Z -6.3333, A 0.000, B 0.000, C 0.000 }
gfCNCPoint5[389] = {X 226.9176, Y 15.5950, Z -6.3333, A 0.000, B 0.000, C 0.000 }
gfCNCPoint5[390] = {X 226.2738, Y 16.2734, Z -6.3333, A 0.000, B 0.000, C 0.000 }
gfCNCPoint5[391] = {X 226.2748, Y 40.9156, Z -6.3333, A 0.000, B 0.000, C 0.000 }
gfCNCPoint5[392] = {X 226.9119, Y 41.5857, Z -6.3333, A 0.000, B 0.000, C 0.000 }
gfCNCPoint5[393] = {X 227.3918, Y 42.3761, Z -6.3333, A 0.000, B 0.000, C 0.000 }
gfCNCPoint5[394] = {X 227.6926, Y 43.2505, Z -6.3333, A 0.000, B 0.000, C 0.000 }
gfCNCPoint5[395] = {X 227.8003, Y 44.1689, Z -6.3333, A 0.000, B 0.000, C 0.000 }
gfCNCPoint5[396] = {X 227.8005, Y 45.0000, Z -6.3333, A 0.000, B 0.000, C 0.000 }
gfCNCPoint5[397] = {X 227.6922, Y 45.9613, Z -6.3333, A 0.000, B 0.000, C 0.000 }
gfCNCPoint5[398] = {X 227.3727, Y 46.8744, Z -6.3333, A 0.000, B 0.000, C 0.000 }
gfCNCPoint5[399] = {X 226.8580, Y 47.6935, Z -6.3333, A 0.000, B 0.000, C 0.000 }
gfCNCPoint5[400] = {X 226.1740, Y 48.3775, Z -6.3333, A 0.000, B 0.000, C 0.000 }
gfCNCPoint5[401] = {X 225.3549, Y 48.8922, Z -6.3333, A 0.000, B 0.000, C 0.000 }
gfCNCPoint5[402] = {X 224.4418, Y 49.2117, Z -6.3333, A 0.000, B 0.000, C 0.000 }
gfCNCPoint5[403] = {X 223.4805, Y 49.3200, Z -6.3333, A 0.000, B 0.000, C 0.000 }
gfCNCPoint5[404] = {X 217.0370, Y 49.3200, Z -6.3333, A 0.000, B 0.000, C 0.000 }
gfCNCPoint5[405] = {X 216.0805, Y 49.2128, Z -6.3333, A 0.000, B 0.000, C 0.000 }
gfCNCPoint5[406] = {X 215.1715, Y 48.8964, Z -6.3333, A 0.000, B 0.000, C 0.000 }
gfCNCPoint5[407] = {X 214.3551, Y 48.3867, Z -6.3333, A 0.000, B 0.000, C 0.000 }
gfCNCPoint5[408] = {X 213.6718, Y 47.7088, Z -6.3333, A 0.000, B 0.000, C 0.000 }
gfCNCPoint5[409] = {X 213.1556, Y 46.8965, Z -6.3333, A 0.000, B 0.000, C 0.000 }
gfCNCPoint5[410] = {X 212.8320, Y 45.9901, Z -6.3333, A 0.000, B 0.000, C 0.000 }
gfCNCPoint5[411] = {X 212.7172, Y 45.0345, Z -6.3333, A 0.000, B 0.000, C 0.000 }
gfCNCPoint5[412] = {X 212.7170, Y 44.1918, Z -6.3333, A 0.000, B 0.000, C 0.000 }
gfCNCPoint5[413] = {X 212.7887, Y 43.4152, Z -6.3333, A 0.000, B 0.000, C 0.000 }
gfCNCPoint5[414] = {X 213.0014, Y 42.6648, Z -6.3333, A 0.000, B 0.000, C 0.000 }
gfCNCPoint5[415] = {X 213.3478, Y 41.9660, Z -6.3333, A 0.000, B 0.000, C 0.000 }
gfCNCPoint5[416] = {X 213.8163, Y 41.3425, Z -6.3333, A 0.000, B 0.000, C 0.000 }
gfCNCPoint5[417] = {X 214.2398, Y 40.8754, Z -6.3333, A 0.000, B 0.000, C 0.000 }
gfCNCPoint5[418] = {X 214.2442, Y 40.3062, Z -6.3333, A 0.000, B 0.000, C 0.000 }
gfCNCPoint5[419] = {X 214.2442, Y 28.5738, Z -6.3333, A 0.000, B 0.000, C 0.000 }
gfCNCPoint5[420] = {X 210.2442, Y 28.5738, Z -6.3333, A 0.000, B 0.000, C 0.000 }
gfCNCPoint5[421] = {X 214.3242, Y 28.5738, Z -6.3333, A 0.000, B 0.000, C 0.000 }
gfCNCPoint5[422] = {X 214.3242, Y 17.4621, Z -6.3333, A 0.000, B 0.000, C 0.000 }
gfCNCPoint5[423] = {X 214.3189, Y 16.7692, Z -6.3333, A 0.000, B 0.000, C 0.000 }
gfCNCPoint5[424] = {X 214.3225, Y 16.2352, Z -6.3333, A 0.000, B 0.000, C 0.000 }
gfCNCPoint5[425] = {X 213.6851, Y 15.5747, Z -6.3333, A 0.000, B 0.000, C 0.000 }
gfCNCPoint5[426] = {X 213.2049, Y 14.7925, Z -6.3333, A 0.000, B 0.000, C 0.000 }
gfCNCPoint5[427] = {X 212.9042, Y 13.9253, Z -6.3333, A 0.000, B 0.000, C 0.000 }
gfCNCPoint5[428] = {X 212.7972, Y 13.0136, Z -6.3333, A 0.000, B 0.000, C 0.000 }
gfCNCPoint5[429] = {X 212.7970, Y 12.1868, Z -6.3333, A 0.000, B 0.000, C 0.000 }
gfCNCPoint5[430] = {X 212.9033, Y 11.2433, Z -6.3333, A 0.000, B 0.000, C 0.000 }
gfCNCPoint5[431] = {X 213.2169, Y 10.3472, Z -6.3333, A 0.000, B 0.000, C 0.000 }
gfCNCPoint5[432] = {X 213.7220, Y 9.5432, Z -6.3333, A 0.000, B 0.000, C 0.000 }
gfCNCPoint5[433] = {X 214.3934, Y 8.8719, Z -6.3333, A 0.000, B 0.000, C 0.000 }
gfCNCPoint5[434] = {X 215.1973, Y 8.3667, Z -6.3333, A 0.000, B 0.000, C 0.000 }
gfCNCPoint5[435] = {X 216.0935, Y 8.0531, Z -6.3333, A 0.000, B 0.000, C 0.000 }
gfCNCPoint5[436] = {X 217.0370, Y 7.9468, Z -6.3333, A 0.000, B 0.000, C 0.000 }
gfCNCPoint5[437] = {X 223.4805, Y 7.9468, Z -6.3333, A 0.000, B 0.000, C 0.000 }
gfCNCPoint5[438] = {X 224.4240, Y 8.0531, Z -6.3333, A 0.000, B 0.000, C 0.000 }
gfCNCPoint5[439] = {X 225.3201, Y 8.3667, Z -6.3333, A 0.000, B 0.000, C 0.000 }
gfCNCPoint5[440] = {X 226.1241, Y 8.8718, Z -6.3333, A 0.000, B 0.000, C 0.000 }
gfCNCPoint5[441] = {X 226.7954, Y 9.5432, Z -6.3333, A 0.000, B 0.000, C 0.000 }
gfCNCPoint5[442] = {X 227.3006, Y 10.3471, Z -6.3333, A 0.000, B 0.000, C 0.000 }
gfCNCPoint5[443] = {X 227.6142, Y 11.2433, Z -6.3333, A 0.000, B 0.000, C 0.000 }
gfCNCPoint5[444] = {X 227.7205, Y 12.1868, Z -6.3333, A 0.000, B 0.000, C 0.000 }
gfCNCPoint5[445] = {X 227.7205, Y 12.9782, Z -6.3333, A 0.000, B 0.000, C 0.000 }
gfCNCPoint5[446] = {X 227.6191, Y 13.8997, Z -6.3333, A 0.000, B 0.000, C 0.000 }
gfCNCPoint5[447] = {X 227.3199, Y 14.7771, Z -6.3333, A 0.000, B 0.000, C 0.000 }
gfCNCPoint5[448] = {X 226.8371, Y 15.5685, Z -6.3333, A 0.000, B 0.000, C 0.000 }
gfCNCPoint5[449] = {X 226.1938, Y 16.2361, Z -6.3333, A 0.000, B 0.000, C 0.000 }
gfCNCPoint5[450] = {X 226.1948, Y 40.9528, Z -6.3333, A 0.000, B 0.000, C 0.000 }
gfCNCPoint5[451] = {X 226.8315, Y 41.6124, Z -6.3333, A 0.000, B 0.000, C 0.000 }
gfCNCPoint5[452] = {X 227.3115, Y 42.3934, Z -6.3333, A 0.000, B 0.000, C 0.000 }
gfCNCPoint5[453] = {X 227.6125, Y 43.2593, Z -6.3333, A 0.000, B 0.000, C 0.000 }
gfCNCPoint5[454] = {X 227.7203, Y 44.1697, Z -6.3333, A 0.000, B 0.000, C 0.000 }
gfCNCPoint5[455] = {X 227.7205, Y 45.0000, Z -6.3333, A 0.000, B 0.000, C 0.000 }
gfCNCPoint5[456] = {X 227.6142, Y 45.9435, Z -6.3333, A 0.000, B 0.000, C 0.000 }
gfCNCPoint5[457] = {X 227.3006, Y 46.8397, Z -6.3333, A 0.000, B 0.000, C 0.000 }
gfCNCPoint5[458] = {X 226.7954, Y 47.6436, Z -6.3333, A 0.000, B 0.000, C 0.000 }
gfCNCPoint5[459] = {X 226.1241, Y 48.3150, Z -6.3333, A 0.000, B 0.000, C 0.000 }
gfCNCPoint5[460] = {X 225.3201, Y 48.8201, Z -6.3333, A 0.000, B 0.000, C 0.000 }
gfCNCPoint5[461] = {X 224.4240, Y 49.1337, Z -6.3333, A 0.000, B 0.000, C 0.000 }
gfCNCPoint5[462] = {X 223.4805, Y 49.2400, Z -6.3333, A 0.000, B 0.000, C 0.000 }
gfCNCPoint5[463] = {X 217.0370, Y 49.2400, Z -6.3333, A 0.000, B 0.000, C 0.000 }
gfCNCPoint5[464] = {X 216.0982, Y 49.1348, Z -6.3333, A 0.000, B 0.000, C 0.000 }
gfCNCPoint5[465] = {X 215.2061, Y 48.8243, Z -6.3333, A 0.000, B 0.000, C 0.000 }
gfCNCPoint5[466] = {X 214.4048, Y 48.3240, Z -6.3333, A 0.000, B 0.000, C 0.000 }
gfCNCPoint5[467] = {X 213.7341, Y 47.6587, Z -6.3333, A 0.000, B 0.000, C 0.000 }
gfCNCPoint5[468] = {X 213.2275, Y 46.8614, Z -6.3333, A 0.000, B 0.000, C 0.000 }
gfCNCPoint5[469] = {X 212.9099, Y 45.9717, Z -6.3333, A 0.000, B 0.000, C 0.000 }
gfCNCPoint5[470] = {X 212.7972, Y 45.0338, Z -6.3333, A 0.000, B 0.000, C 0.000 }
gfCNCPoint5[471] = {X 212.7970, Y 44.1918, Z -6.3333, A 0.000, B 0.000, C 0.000 }
gfCNCPoint5[472] = {X 212.8674, Y 43.4298, Z -6.3333, A 0.000, B 0.000, C 0.000 }
gfCNCPoint5[473] = {X 213.0760, Y 42.6936, Z -6.3333, A 0.000, B 0.000, C 0.000 }
gfCNCPoint5[474] = {X 213.4159, Y 42.0080, Z -6.3333, A 0.000, B 0.000, C 0.000 }
gfCNCPoint5[475] = {X 213.8756, Y 41.3962, Z -6.3333, A 0.000, B 0.000, C 0.000 }
gfCNCPoint5[476] = {X 214.3196, Y 40.9065, Z -6.3333, A 0.000, B 0.000, C 0.000 }
gfCNCPoint5[477] = {X 214.3242, Y 40.3065, Z -6.3333, A 0.000, B 0.000, C 0.000 }
gfCNCPoint5[478] = {X 214.3242, Y 28.5738, Z -6.3333, A 0.000, B 0.000, C 0.000 }
gfCNCPoint5[479] = {X 210.3242, Y 28.5738, Z -6.3333, A 0.000, B 0.000, C 0.000 }
gfCNCPoint5[480] = {X 214.4042, Y 28.5738, Z -6.3333, A 0.000, B 0.000, C 0.000 }
gfCNCPoint5[481] = {X 214.4042, Y 17.4618, Z -6.3333, A 0.000, B 0.000, C 0.000 }
gfCNCPoint5[482] = {X 214.3989, Y 16.7691, Z -6.3333, A 0.000, B 0.000, C 0.000 }
gfCNCPoint5[483] = {X 214.4027, Y 16.1977, Z -6.3333, A 0.000, B 0.000, C 0.000 }
gfCNCPoint5[484] = {X 213.7658, Y 15.5479, Z -6.3333, A 0.000, B 0.000, C 0.000 }
gfCNCPoint5[485] = {X 213.2853, Y 14.7752, Z -6.3333, A 0.000, B 0.000, C 0.000 }
gfCNCPoint5[486] = {X 212.9843, Y 13.9166, Z -6.3333, A 0.000, B 0.000, C 0.000 }
gfCNCPoint5[487] = {X 212.8772, Y 13.0130, Z -6.3333, A 0.000, B 0.000, C 0.000 }
gfCNCPoint5[488] = {X 212.8770, Y 12.1868, Z -6.3333, A 0.000, B 0.000, C 0.000 }
gfCNCPoint5[489] = {X 212.9813, Y 11.2611, Z -6.3333, A 0.000, B 0.000, C 0.000 }
gfCNCPoint5[490] = {X 213.2890, Y 10.3819, Z -6.3333, A 0.000, B 0.000, C 0.000 }
gfCNCPoint5[491] = {X 213.7846, Y 9.5931, Z -6.3333, A 0.000, B 0.000, C 0.000 }
gfCNCPoint5[492] = {X 214.4433, Y 8.9344, Z -6.3333, A 0.000, B 0.000, C 0.000 }
gfCNCPoint5[493] = {X 215.2321, Y 8.4388, Z -6.3333, A 0.000, B 0.000, C 0.000 }
gfCNCPoint5[494] = {X 216.1113, Y 8.1311, Z -6.3333, A 0.000, B 0.000, C 0.000 }
gfCNCPoint5[495] = {X 217.0370, Y 8.0268, Z -6.3333, A 0.000, B 0.000, C 0.000 }
gfCNCPoint5[496] = {X 223.4805, Y 8.0268, Z -6.3333, A 0.000, B 0.000, C 0.000 }
gfCNCPoint5[497] = {X 224.4062, Y 8.1311, Z -6.3333, A 0.000, B 0.000, C 0.000 }
gfCNCPoint5[498] = {X 225.2854, Y 8.4388, Z -6.3333, A 0.000, B 0.000, C 0.000 }
gfCNCPoint5[499] = {X 226.0742, Y 8.9344, Z -6.3333, A 0.000, B 0.000, C 0.000 }
gfCNCPoint5[500] = {X 226.7329, Y 9.5931, Z -6.3333, A 0.000, B 0.000, C 0.000 }
gfCNCPoint5[501] = {X 227.2285, Y 10.3819, Z -6.3333, A 0.000, B 0.000, C 0.000 }
gfCNCPoint5[502] = {X 227.5362, Y 11.2611, Z -6.3333, A 0.000, B 0.000, C 0.000 }
gfCNCPoint5[503] = {X 227.6405, Y 12.1868, Z -6.3333, A 0.000, B 0.000, C 0.000 }
gfCNCPoint5[504] = {X 227.6405, Y 12.9782, Z -6.3333, A 0.000, B 0.000, C 0.000 }
gfCNCPoint5[505] = {X 227.5390, Y 13.8914, Z -6.3333, A 0.000, B 0.000, C 0.000 }
gfCNCPoint5[506] = {X 227.2395, Y 14.7601, Z -6.3333, A 0.000, B 0.000, C 0.000 }
gfCNCPoint5[507] = {X 226.7566, Y 15.5418, Z -6.3333, A 0.000, B 0.000, C 0.000 }
gfCNCPoint5[508] = {X 226.1138, Y 16.1984, Z -6.3333, A 0.000, B 0.000, C 0.000 }
gfCNCPoint5[509] = {X 226.1148, Y 40.9905, Z -6.3333, A 0.000, B 0.000, C 0.000 }
gfCNCPoint5[510] = {X 226.7510, Y 41.6393, Z -6.3333, A 0.000, B 0.000, C 0.000 }
gfCNCPoint5[511] = {X 227.2312, Y 42.4108, Z -6.3333, A 0.000, B 0.000, C 0.000 }
gfCNCPoint5[512] = {X 227.5324, Y 43.2681, Z -6.3333, A 0.000, B 0.000, C 0.000 }
gfCNCPoint5[513] = {X 227.6403, Y 44.1704, Z -6.3333, A 0.000, B 0.000, C 0.000 }
gfCNCPoint5[514] = {X 227.6405, Y 45.0000, Z -6.3333, A 0.000, B 0.000, C 0.000 }
gfCNCPoint5[515] = {X 227.5362, Y 45.9257, Z -6.3333, A 0.000, B 0.000, C 0.000 }
gfCNCPoint5[516] = {X 227.2285, Y 46.8050, Z -6.3333, A 0.000, B 0.000, C 0.000 }
gfCNCPoint5[517] = {X 226.7329, Y 47.5937, Z -6.3333, A 0.000, B 0.000, C 0.000 }
gfCNCPoint5[518] = {X 226.0742, Y 48.2524, Z -6.3333, A 0.000, B 0.000, C 0.000 }
gfCNCPoint5[519] = {X 225.2854, Y 48.7480, Z -6.3333, A 0.000, B 0.000, C 0.000 }
gfCNCPoint5[520] = {X 224.4062, Y 49.0557, Z -6.3333, A 0.000, B 0.000, C 0.000 }
gfCNCPoint5[521] = {X 223.4805, Y 49.1600, Z -6.3333, A 0.000, B 0.000, C 0.000 }
gfCNCPoint5[522] = {X 217.0370, Y 49.1600, Z -6.3333, A 0.000, B 0.000, C 0.000 }
gfCNCPoint5[523] = {X 216.1160, Y 49.0568, Z -6.3333, A 0.000, B 0.000, C 0.000 }
gfCNCPoint5[524] = {X 215.2406, Y 48.7521, Z -6.3333, A 0.000, B 0.000, C 0.000 }
gfCNCPoint5[525] = {X 214.4544, Y 48.2613, Z -6.3333, A 0.000, B 0.000, C 0.000 }
gfCNCPoint5[526] = {X 213.7965, Y 47.6085, Z -6.3333, A 0.000, B 0.000, C 0.000 }
gfCNCPoint5[527] = {X 213.2993, Y 46.8263, Z -6.3333, A 0.000, B 0.000, C 0.000 }
gfCNCPoint5[528] = {X 212.9877, Y 45.9534, Z -6.3333, A 0.000, B 0.000, C 0.000 }
gfCNCPoint5[529] = {X 212.8771, Y 45.0332, Z -6.3333, A 0.000, B 0.000, C 0.000 }
gfCNCPoint5[530] = {X 212.8770, Y 44.1918, Z -6.3333, A 0.000, B 0.000, C 0.000 }
gfCNCPoint5[531] = {X 212.9460, Y 43.4445, Z -6.3333, A 0.000, B 0.000, C 0.000 }
gfCNCPoint5[532] = {X 213.1507, Y 42.7224, Z -6.3333, A 0.000, B 0.000, C 0.000 }
gfCNCPoint5[533] = {X 213.4840, Y 42.0500, Z -6.3333, A 0.000, B 0.000, C 0.000 }
gfCNCPoint5[534] = {X 213.9349, Y 41.4499, Z -6.3333, A 0.000, B 0.000, C 0.000 }
gfCNCPoint5[535] = {X 214.3993, Y 40.9376, Z -6.3333, A 0.000, B 0.000, C 0.000 }
gfCNCPoint5[536] = {X 214.4042, Y 40.3068, Z -6.3333, A 0.000, B 0.000, C 0.000 }
gfCNCPoint5[537] = {X 214.4042, Y 28.5738, Z -6.3333, A 0.000, B 0.000, C 0.000 }
gfCNCPoint5[538] = {X 210.4042, Y 28.5738, Z -6.3333, A 0.000, B 0.000, C 0.000 }
gfCNCPoint5[539] = {X 214.4842, Y 28.5738, Z -6.3333, A 0.000, B 0.000, C 0.000 }
gfCNCPoint5[540] = {X 214.4842, Y 17.4614, Z -6.3333, A 0.000, B 0.000, C 0.000 }
gfCNCPoint5[541] = {X 214.4789, Y 16.7691, Z -6.3333, A 0.000, B 0.000, C 0.000 }
gfCNCPoint5[542] = {X 214.4830, Y 16.1598, Z -6.3333, A 0.000, B 0.000, C 0.000 }
gfCNCPoint5[543] = {X 214.4250, Y 16.1123, Z -6.3333, A 0.000, B 0.000, C 0.000 }
gfCNCPoint5[544] = {X 214.3678, Y 16.0637, Z -6.3333, A 0.000, B 0.000, C 0.000 }
gfCNCPoint5[545] = {X 213.7775, Y 15.4320, Z -6.3333, A 0.000, B 0.000, C 0.000 }
gfCNCPoint5[546] = {X 213.3336, Y 14.6901, Z -6.3333, A 0.000, B 0.000, C 0.000 }
gfCNCPoint5[547] = {X 213.0560, Y 13.8712, Z -6.3333, A 0.000, B 0.000, C 0.000 }
gfCNCPoint5[548] = {X 212.9572, Y 13.0123, Z -6.3333, A 0.000, B 0.000, C 0.000 }
gfCNCPoint5[549] = {X 212.9570, Y 12.1868, Z -6.3333, A 0.000, B 0.000, C 0.000 }
gfCNCPoint5[550] = {X 213.0593, Y 11.2789, Z -6.3333, A 0.000, B 0.000, C 0.000 }
gfCNCPoint5[551] = {X 213.3611, Y 10.4166, Z -6.3333, A 0.000, B 0.000, C 0.000 }
gfCNCPoint5[552] = {X 213.8471, Y 9.6430, Z -6.3333, A 0.000, B 0.000, C 0.000 }
gfCNCPoint5[553] = {X 214.4932, Y 8.9969, Z -6.3333, A 0.000, B 0.000, C 0.000 }
gfCNCPoint5[554] = {X 215.2668, Y 8.5109, Z -6.3333, A 0.000, B 0.000, C 0.000 }
gfCNCPoint5[555] = {X 216.1291, Y 8.2091, Z -6.3333, A 0.000, B 0.000, C 0.000 }
gfCNCPoint5[556] = {X 217.0370, Y 8.1068, Z -6.3333, A 0.000, B 0.000, C 0.000 }
gfCNCPoint5[557] = {X 223.4805, Y 8.1068, Z -6.3333, A 0.000, B 0.000, C 0.000 }
gfCNCPoint5[558] = {X 224.3884, Y 8.2091, Z -6.3333, A 0.000, B 0.000, C 0.000 }
gfCNCPoint5[559] = {X 225.2507, Y 8.5109, Z -6.3333, A 0.000, B 0.000, C 0.000 }
gfCNCPoint5[560] = {X 226.0243, Y 8.9969, Z -6.3333, A 0.000, B 0.000, C 0.000 }
gfCNCPoint5[561] = {X 226.6704, Y 9.6430, Z -6.3333, A 0.000, B 0.000, C 0.000 }
gfCNCPoint5[562] = {X 227.1564, Y 10.4166, Z -6.3333, A 0.000, B 0.000, C 0.000 }
gfCNCPoint5[563] = {X 227.4582, Y 11.2789, Z -6.3333, A 0.000, B 0.000, C 0.000 }
gfCNCPoint5[564] = {X 227.5605, Y 12.1868, Z -6.3333, A 0.000, B 0.000, C 0.000 }
gfCNCPoint5[565] = {X 227.5605, Y 12.9782, Z -6.3333, A 0.000, B 0.000, C 0.000 }
gfCNCPoint5[566] = {X 227.4588, Y 13.8830, Z -6.3333, A 0.000, B 0.000, C 0.000 }
gfCNCPoint5[567] = {X 227.1590, Y 14.7428, Z -6.3333, A 0.000, B 0.000, C 0.000 }
gfCNCPoint5[568] = {X 226.6760, Y 15.5147, Z -6.3333, A 0.000, B 0.000, C 0.000 }
gfCNCPoint5[569] = {X 226.0338, Y 16.1603, Z -6.3333, A 0.000, B 0.000, C 0.000 }
gfCNCPoint5[570] = {X 226.0348, Y 41.0283, Z -6.3333, A 0.000, B 0.000, C 0.000 }
gfCNCPoint5[571] = {X 226.1411, Y 41.1157, Z -6.3333, A 0.000, B 0.000, C 0.000 }
gfCNCPoint5[572] = {X 226.7344, Y 41.7474, Z -6.3333, A 0.000, B 0.000, C 0.000 }
gfCNCPoint5[573] = {X 227.1808, Y 42.4901, Z -6.3333, A 0.000, B 0.000, C 0.000 }
gfCNCPoint5[574] = {X 227.4603, Y 43.3104, Z -6.3333, A 0.000, B 0.000, C 0.000 }
gfCNCPoint5[575] = {X 227.5603, Y 44.1712, Z -6.3333, A 0.000, B 0.000, C 0.000 }
gfCNCPoint5[576] = {X 227.5605, Y 45.0000, Z -6.3333, A 0.000, B 0.000, C 0.000 }
gfCNCPoint5[577] = {X 227.4582, Y 45.9079, Z -6.3333, A 0.000, B 0.000, C 0.000 }
gfCNCPoint5[578] = {X 227.1564, Y 46.7702, Z -6.3333, A 0.000, B 0.000, C 0.000 }
gfCNCPoint5[579] = {X 226.6704, Y 47.5438, Z -6.3333, A 0.000, B 0.000, C 0.000 }
gfCNCPoint5[580] = {X 226.0243, Y 48.1899, Z -6.3333, A 0.000, B 0.000, C 0.000 }
gfCNCPoint5[581] = {X 225.2507, Y 48.6760, Z -6.3333, A 0.000, B 0.000, C 0.000 }
gfCNCPoint5[582] = {X 224.3884, Y 48.9777, Z -6.3333, A 0.000, B 0.000, C 0.000 }
gfCNCPoint5[583] = {X 223.4805, Y 49.0800, Z -6.3333, A 0.000, B 0.000, C 0.000 }
gfCNCPoint5[584] = {X 217.0370, Y 49.0800, Z -6.3333, A 0.000, B 0.000, C 0.000 }
gfCNCPoint5[585] = {X 216.1337, Y 48.9787, Z -6.3333, A 0.000, B 0.000, C 0.000 }
gfCNCPoint5[586] = {X 215.2752, Y 48.6800, Z -6.3333, A 0.000, B 0.000, C 0.000 }
gfCNCPoint5[587] = {X 214.5041, Y 48.1986, Z -6.3333, A 0.000, B 0.000, C 0.000 }
gfCNCPoint5[588] = {X 213.8588, Y 47.5584, Z -6.3333, A 0.000, B 0.000, C 0.000 }
gfCNCPoint5[589] = {X 213.3712, Y 46.7912, Z -6.3333, A 0.000, B 0.000, C 0.000 }
gfCNCPoint5[590] = {X 213.0656, Y 45.9351, Z -6.3333, A 0.000, B 0.000, C 0.000 }
gfCNCPoint5[591] = {X 212.9571, Y 45.0325, Z -6.3333, A 0.000, B 0.000, C 0.000 }
gfCNCPoint5[592] = {X 212.9570, Y 44.1918, Z -6.3333, A 0.000, B 0.000, C 0.000 }
gfCNCPoint5[593] = {X 213.0247, Y 43.4591, Z -6.3333, A 0.000, B 0.000, C 0.000 }
gfCNCPoint5[594] = {X 213.2253, Y 42.7512, Z -6.3333, A 0.000, B 0.000, C 0.000 }
gfCNCPoint5[595] = {X 213.5521, Y 42.0919, Z -6.3333, A 0.000, B 0.000, C 0.000 }
gfCNCPoint5[596] = {X 213.9941, Y 41.5037, Z -6.3333, A 0.000, B 0.000, C 0.000 }
gfCNCPoint5[597] = {X 214.4791, Y 40.9687, Z -6.3333, A 0.000, B 0.000, C 0.000 }
gfCNCPoint5[598] = {X 214.4842, Y 40.3072, Z -6.3333, A 0.000, B 0.000, C 0.000 }
gfCNCPoint5[599] = {X 214.4842, Y 28.5738, Z -6.3333, A 0.000, B 0.000, C 0.000 }
gfCNCPoint5[600] = {X 210.4842, Y 28.5738, Z -6.3333, A 0.000, B 0.000, C 0.000 }
gfCNCPoint5[601] = {X 214.5642, Y 28.5738, Z -6.3333, A 0.000, B 0.000, C 0.000 }
gfCNCPoint5[602] = {X 214.5642, Y 17.4611, Z -6.3333, A 0.000, B 0.000, C 0.000 }
gfCNCPoint5[603] = {X 214.5589, Y 16.7687, Z -6.3333, A 0.000, B 0.000, C 0.000 }
gfCNCPoint5[604] = {X 214.5583, Y 16.1870, Z -6.3333, A 0.000, B 0.000, C 0.000 }
gfCNCPoint5[605] = {X 214.5756, Y 16.1310, Z -6.3333, A 0.000, B 0.000, C 0.000 }
gfCNCPoint5[606] = {X 214.4971, Y 16.0681, Z -6.3333, A 0.000, B 0.000, C 0.000 }
gfCNCPoint5[607] = {X 214.4201, Y 16.0032, Z -6.3333, A 0.000, B 0.000, C 0.000 }
gfCNCPoint5[608] = {X 213.8364, Y 15.3772, Z -6.3333, A 0.000, B 0.000, C 0.000 }
gfCNCPoint5[609] = {X 213.3992, Y 14.6412, Z -6.3333, A 0.000, B 0.000, C 0.000 }
gfCNCPoint5[610] = {X 213.1286, Y 13.8291, Z -6.3333, A 0.000, B 0.000, C 0.000 }
gfCNCPoint5[611] = {X 213.0370, Y 12.9780, Z -6.3333, A 0.000, B 0.000, C 0.000 }
gfCNCPoint5[612] = {X 213.0370, Y 12.1868, Z -6.3333, A 0.000, B 0.000, C 0.000 }
gfCNCPoint5[613] = {X 213.1373, Y 11.2967, Z -6.3333, A 0.000, B 0.000, C 0.000 }
gfCNCPoint5[614] = {X 213.4331, Y 10.4513, Z -6.3333, A 0.000, B 0.000, C 0.000 }
gfCNCPoint5[615] = {X 213.9097, Y 9.6929, Z -6.3333, A 0.000, B 0.000, C 0.000 }
gfCNCPoint5[616] = {X 214.5431, Y 9.0595, Z -6.3333, A 0.000, B 0.000, C 0.000 }
gfCNCPoint5[617] = {X 215.3015, Y 8.5829, Z -6.3333, A 0.000, B 0.000, C 0.000 }
gfCNCPoint5[618] = {X 216.1469, Y 8.2871, Z -6.3333, A 0.000, B 0.000, C 0.000 }
gfCNCPoint5[619] = {X 217.0370, Y 8.1868, Z -6.3333, A 0.000, B 0.000, C 0.000 }
gfCNCPoint5[620] = {X 223.4805, Y 8.1868, Z -6.3333, A 0.000, B 0.000, C 0.000 }
gfCNCPoint5[621] = {X 224.3706, Y 8.2871, Z -6.3333, A 0.000, B 0.000, C 0.000 }
gfCNCPoint5[622] = {X 225.2160, Y 8.5829, Z -6.3333, A 0.000, B 0.000, C 0.000 }
gfCNCPoint5[623] = {X 225.9744, Y 9.0595, Z -6.3333, A 0.000, B 0.000, C 0.000 }
gfCNCPoint5[624] = {X 226.6078, Y 9.6929, Z -6.3333, A 0.000, B 0.000, C 0.000 }
gfCNCPoint5[625] = {X 227.0844, Y 10.4513, Z -6.3333, A 0.000, B 0.000, C 0.000 }
gfCNCPoint5[626] = {X 227.3802, Y 11.2967, Z -6.3333, A 0.000, B 0.000, C 0.000 }
gfCNCPoint5[627] = {X 227.4805, Y 12.1868, Z -6.3333, A 0.000, B 0.000, C 0.000 }
gfCNCPoint5[628] = {X 227.4803, Y 13.0192, Z -6.3333, A 0.000, B 0.000, C 0.000 }
gfCNCPoint5[629] = {X 227.3717, Y 13.9046, Z -6.3333, A 0.000, B 0.000, C 0.000 }
gfCNCPoint5[630] = {X 227.0696, Y 14.7439, Z -6.3333, A 0.000, B 0.000, C 0.000 }
gfCNCPoint5[631] = {X 226.5890, Y 15.4954, Z -6.3333, A 0.000, B 0.000, C 0.000 }
gfCNCPoint5[632] = {X 225.9538, Y 16.1217, Z -6.3333, A 0.000, B 0.000, C 0.000 }
gfCNCPoint5[633] = {X 225.9548, Y 41.0662, Z -6.3333, A 0.000, B 0.000, C 0.000 }
gfCNCPoint5[634] = {X 226.0935, Y 41.1802, Z -6.3333, A 0.000, B 0.000, C 0.000 }
gfCNCPoint5[635] = {X 226.6788, Y 41.8066, Z -6.3333, A 0.000, B 0.000, C 0.000 }
gfCNCPoint5[636] = {X 227.1173, Y 42.5433, Z -6.3333, A 0.000, B 0.000, C 0.000 }
gfCNCPoint5[637] = {X 227.3886, Y 43.3565, Z -6.3333, A 0.000, B 0.000, C 0.000 }
gfCNCPoint5[638] = {X 227.4805, Y 44.2089, Z -6.3333, A 0.000, B 0.000, C 0.000 }
gfCNCPoint5[639] = {X 227.4805, Y 45.0000, Z -6.3333, A 0.000, B 0.000, C 0.000 }
gfCNCPoint5[640] = {X 227.3802, Y 45.8901, Z -6.3333, A 0.000, B 0.000, C 0.000 }
gfCNCPoint5[641] = {X 227.0844, Y 46.7355, Z -6.3333, A 0.000, B 0.000, C 0.000 }
gfCNCPoint5[642] = {X 226.6078, Y 47.4940, Z -6.3333, A 0.000, B 0.000, C 0.000 }
gfCNCPoint5[643] = {X 225.9744, Y 48.1273, Z -6.3333, A 0.000, B 0.000, C 0.000 }
gfCNCPoint5[644] = {X 225.2160, Y 48.6039, Z -6.3333, A 0.000, B 0.000, C 0.000 }
gfCNCPoint5[645] = {X 224.3706, Y 48.8997, Z -6.3333, A 0.000, B 0.000, C 0.000 }
gfCNCPoint5[646] = {X 223.4805, Y 49.0000, Z -6.3333, A 0.000, B 0.000, C 0.000 }
gfCNCPoint5[647] = {X 217.0370, Y 49.0000, Z -6.3333, A 0.000, B 0.000, C 0.000 }
gfCNCPoint5[648] = {X 216.1469, Y 48.8997, Z -6.3333, A 0.000, B 0.000, C 0.000 }
gfCNCPoint5[649] = {X 215.3015, Y 48.6039, Z -6.3333, A 0.000, B 0.000, C 0.000 }
gfCNCPoint5[650] = {X 214.5430, Y 48.1273, Z -6.3333, A 0.000, B 0.000, C 0.000 }
gfCNCPoint5[651] = {X 213.9097, Y 47.4939, Z -6.3333, A 0.000, B 0.000, C 0.000 }
gfCNCPoint5[652] = {X 213.4331, Y 46.7355, Z -6.3333, A 0.000, B 0.000, C 0.000 }
gfCNCPoint5[653] = {X 213.1373, Y 45.8901, Z -6.3333, A 0.000, B 0.000, C 0.000 }
gfCNCPoint5[654] = {X 213.0370, Y 45.0000, Z -6.3333, A 0.000, B 0.000, C 0.000 }
gfCNCPoint5[655] = {X 213.0370, Y 44.1918, Z -6.3333, A 0.000, B 0.000, C 0.000 }
gfCNCPoint5[656] = {X 213.1546, Y 43.2386, Z -6.3333, A 0.000, B 0.000, C 0.000 }
gfCNCPoint5[657] = {X 213.5003, Y 42.3426, Z -6.3333, A 0.000, B 0.000, C 0.000 }
gfCNCPoint5[658] = {X 214.0534, Y 41.5574, Z -6.3333, A 0.000, B 0.000, C 0.000 }
gfCNCPoint5[659] = {X 214.5589, Y 40.9999, Z -6.3333, A 0.000, B 0.000, C 0.000 }
gfCNCPoint5[660] = {X 214.5642, Y 40.3075, Z -6.3333, A 0.000, B 0.000, C 0.000 }
gfCNCPoint5[661] = {X 214.5642, Y 28.5738, Z -6.3333, A 0.000, B 0.000, C 0.000 }
gfCNCPoint5[662] = {X 210.4842, Y 28.5738, Z -6.3333, A 0.000, B 0.000, C 0.000 }
gfCNCPoint5[663] = {X 210.4842, Y 28.5738, Z -3.3333, A 0.000, B 0.000, C 0.000 }
gfCNCPoint5[664] = {X 210.4842, Y 28.5738, Z 11.0000, A 0.000, B 0.000, C 0.000 }
gfCNCPoint5[665] = {X 273.6045, Y 28.5936, Z 11.0000, A 0.000, B 0.000, C 0.000 }
gfCNCPoint5[666] = {X 273.6045, Y 28.5936, Z -3.3333, A 0.000, B 0.000, C 0.000 }
gfCNCPoint5[667] = {X 273.6045, Y 28.5936, Z -6.3333, A 0.000, B 0.000, C 0.000 }
gfCNCPoint5[668] = {X 269.5245, Y 28.5936, Z -6.3333, A 0.000, B 0.000, C 0.000 }
gfCNCPoint5[669] = {X 269.5245, Y 40.9139, Z -6.3333, A 0.000, B 0.000, C 0.000 }
gfCNCPoint5[670] = {X 269.5379, Y 40.9249, Z -6.3333, A 0.000, B 0.000, C 0.000 }
gfCNCPoint5[671] = {X 270.1701, Y 41.5944, Z -6.3333, A 0.000, B 0.000, C 0.000 }
gfCNCPoint5[672] = {X 270.6461, Y 42.3827, Z -6.3333, A 0.000, B 0.000, C 0.000 }
gfCNCPoint5[673] = {X 270.9442, Y 43.2539, Z -6.3333, A 0.000, B 0.000, C 0.000 }
gfCNCPoint5[674] = {X 271.0508, Y 44.1686, Z -6.3333, A 0.000, B 0.000, C 0.000 }
gfCNCPoint5[675] = {X 271.0510, Y 45.0000, Z -6.3333, A 0.000, B 0.000, C 0.000 }
gfCNCPoint5[676] = {X 270.9427, Y 45.9613, Z -6.3333, A 0.000, B 0.000, C 0.000 }
gfCNCPoint5[677] = {X 270.6232, Y 46.8744, Z -6.3333, A 0.000, B 0.000, C 0.000 }
gfCNCPoint5[678] = {X 270.1085, Y 47.6935, Z -6.3333, A 0.000, B 0.000, C 0.000 }
gfCNCPoint5[679] = {X 269.4245, Y 48.3775, Z -6.3333, A 0.000, B 0.000, C 0.000 }
gfCNCPoint5[680] = {X 268.6054, Y 48.8922, Z -6.3333, A 0.000, B 0.000, C 0.000 }
gfCNCPoint5[681] = {X 267.6923, Y 49.2117, Z -6.3333, A 0.000, B 0.000, C 0.000 }
gfCNCPoint5[682] = {X 266.7310, Y 49.3200, Z -6.3333, A 0.000, B 0.000, C 0.000 }
gfCNCPoint5[683] = {X 260.2876, Y 49.3200, Z -6.3333, A 0.000, B 0.000, C 0.000 }
gfCNCPoint5[684] = {X 259.3310, Y 49.2128, Z -6.3333, A 0.000, B 0.000, C 0.000 }
gfCNCPoint5[685] = {X 258.4219, Y 48.8963, Z -6.3333, A 0.000, B 0.000, C 0.000 }
gfCNCPoint5[686] = {X 257.6054, Y 48.3865, Z -6.3333, A 0.000, B 0.000, C 0.000 }
gfCNCPoint5[687] = {X 256.9221, Y 47.7085, Z -6.3333, A 0.000, B 0.000, C 0.000 }
gfCNCPoint5[688] = {X 256.4059, Y 46.8960, Z -6.3333, A 0.000, B 0.000, C 0.000 }
gfCNCPoint5[689] = {X 256.0824, Y 45.9894, Z -6.3333, A 0.000, B 0.000, C 0.000 }
gfCNCPoint5[690] = {X 255.9677, Y 45.0336, Z -6.3333, A 0.000, B 0.000, C 0.000 }
gfCNCPoint5[691] = {X 255.9680, Y 44.1494, Z -6.3333, A 0.000, B 0.000, C 0.000 }
gfCNCPoint5[692] = {X 256.0784, Y 43.2364, Z -6.3333, A 0.000, B 0.000, C 0.000 }
gfCNCPoint5[693] = {X 256.3796, Y 42.3675, Z -6.3333, A 0.000, B 0.000, C 0.000 }
gfCNCPoint5[694] = {X 256.8579, Y 41.5821, Z -6.3333, A 0.000, B 0.000, C 0.000 }
gfCNCPoint5[695] = {X 257.4915, Y 40.9157, Z -6.3333, A 0.000, B 0.000, C 0.000 }
gfCNCPoint5[696] = {X 257.4915, Y 34.4738, Z -6.3333, A 0.000, B 0.000, C 0.000 }
gfCNCPoint5[697] = {X 254.7683, Y 34.4738, Z -6.3333, A 0.000, B 0.000, C 0.000 }
gfCNCPoint5[698] = {X 250.4839, Y 42.8191, Z -6.3333, A 0.000, B 0.000, C 0.000 }
gfCNCPoint5[699] = {X 250.6527, Y 43.4865, Z -6.3333, A 0.000, B 0.000, C 0.000 }
gfCNCPoint5[700] = {X 250.7134, Y 44.1723, Z -6.3333, A 0.000, B 0.000, C 0.000 }
gfCNCPoint5[701] = {X 250.7136, Y 45.0000, Z -6.3333, A 0.000, B 0.000, C 0.000 }
gfCNCPoint5[702] = {X 250.6052, Y 45.9613, Z -6.3333, A 0.000, B 0.000, C 0.000 }
gfCNCPoint5[703] = {X 250.2857, Y 46.8744, Z -6.3333, A 0.000, B 0.000, C 0.000 }
gfCNCPoint5[704] = {X 249.7711, Y 47.6935, Z -6.3333, A 0.000, B 0.000, C 0.000 }
gfCNCPoint5[705] = {X 249.0870, Y 48.3775, Z -6.3333, A 0.000, B 0.000, C 0.000 }
gfCNCPoint5[706] = {X 248.2679, Y 48.8922, Z -6.3333, A 0.000, B 0.000, C 0.000 }
gfCNCPoint5[707] = {X 247.3548, Y 49.2117, Z -6.3333, A 0.000, B 0.000, C 0.000 }
gfCNCPoint5[708] = {X 246.3936, Y 49.3200, Z -6.3333, A 0.000, B 0.000, C 0.000 }
gfCNCPoint5[709] = {X 239.8075, Y 49.3200, Z -6.3333, A 0.000, B 0.000, C 0.000 }
gfCNCPoint5[710] = {X 238.8462, Y 49.2117, Z -6.3333, A 0.000, B 0.000, C 0.000 }
gfCNCPoint5[711] = {X 237.9331, Y 48.8922, Z -6.3333, A 0.000, B 0.000, C 0.000 }
gfCNCPoint5[712] = {X 237.1141, Y 48.3775, Z -6.3333, A 0.000, B 0.000, C 0.000 }
gfCNCPoint5[713] = {X 236.4300, Y 47.6935, Z -6.3333, A 0.000, B 0.000, C 0.000 }
gfCNCPoint5[714] = {X 235.9153, Y 46.8745, Z -6.3333, A 0.000, B 0.000, C 0.000 }
gfCNCPoint5[715] = {X 235.5958, Y 45.9614, Z -6.3333, A 0.000, B 0.000, C 0.000 }
gfCNCPoint5[716] = {X 235.4875, Y 45.0001, Z -6.3333, A 0.000, B 0.000, C 0.000 }
gfCNCPoint5[717] = {X 235.4879, Y 44.1494, Z -6.3333, A 0.000, B 0.000, C 0.000 }
gfCNCPoint5[718] = {X 235.5856, Y 43.2935, Z -6.3333, A 0.000, B 0.000, C 0.000 }
gfCNCPoint5[719] = {X 235.8511, Y 42.4740, Z -6.3333, A 0.000, B 0.000, C 0.000 }
gfCNCPoint5[720] = {X 236.2739, Y 41.7236, Z -6.3333, A 0.000, B 0.000, C 0.000 }
gfCNCPoint5[721] = {X 236.8373, Y 41.0719, Z -6.3333, A 0.000, B 0.000, C 0.000 }
gfCNCPoint5[722] = {X 237.5187, Y 40.5449, Z -6.3333, A 0.000, B 0.000, C 0.000 }
gfCNCPoint5[723] = {X 238.2911, Y 40.1637, Z -6.3333, A 0.000, B 0.000, C 0.000 }
gfCNCPoint5[724] = {X 242.2800, Y 32.3559, Z -6.3333, A 0.000, B 0.000, C 0.000 }
gfCNCPoint5[725] = {X 241.1100, Y 31.5694, Z -6.3333, A 0.000, B 0.000, C 0.000 }
gfCNCPoint5[726] = {X 240.0467, Y 30.6435, Z -6.3333, A 0.000, B 0.000, C 0.000 }
gfCNCPoint5[727] = {X 239.1068, Y 29.5927, Z -6.3333, A 0.000, B 0.000, C 0.000 }
gfCNCPoint5[728] = {X 238.3048, Y 28.4332, Z -6.3333, A 0.000, B 0.000, C 0.000 }
gfCNCPoint5[729] = {X 237.6532, Y 27.1830, Z -6.3333, A 0.000, B 0.000, C 0.000 }
gfCNCPoint5[730] = {X 237.1619, Y 25.8615, Z -6.3333, A 0.000, B 0.000, C 0.000 }
gfCNCPoint5[731] = {X 236.7418, Y 24.0500, Z -6.3333, A 0.000, B 0.000, C 0.000 }
gfCNCPoint5[732] = {X 236.5276, Y 22.2029, Z -6.3333, A 0.000, B 0.000, C 0.000 }
gfCNCPoint5[733] = {X 236.5223, Y 20.3433, Z -6.3333, A 0.000, B 0.000, C 0.000 }
gfCNCPoint5[734] = {X 236.7257, Y 18.4950, Z -6.3333, A 0.000, B 0.000, C 0.000 }
gfCNCPoint5[735] = {X 237.1355, Y 16.6811, Z -6.3333, A 0.000, B 0.000, C 0.000 }
gfCNCPoint5[736] = {X 237.7059, Y 15.1053, Z -6.3333, A 0.000, B 0.000, C 0.000 }
gfCNCPoint5[737] = {X 238.4930, Y 13.6258, Z -6.3333, A 0.000, B 0.000, C 0.000 }
gfCNCPoint5[738] = {X 239.4809, Y 12.2720, Z -6.3333, A 0.000, B 0.000, C 0.000 }
gfCNCPoint5[739] = {X 240.6499, Y 11.0712, Z -6.3333, A 0.000, B 0.000, C 0.000 }
gfCNCPoint5[740] = {X 241.9767, Y 10.0473, Z -6.3333, A 0.000, B 0.000, C 0.000 }
gfCNCPoint5[741] = {X 243.4346, Y 9.2208, Z -6.3333, A 0.000, B 0.000, C 0.000 }
gfCNCPoint5[742] = {X 244.9945, Y 8.6083, Z -6.3333, A 0.000, B 0.000, C 0.000 }
gfCNCPoint5[743] = {X 246.6252, Y 8.2219, Z -6.3333, A 0.000, B 0.000, C 0.000 }
gfCNCPoint5[744] = {X 248.7221, Y 7.9504, Z -6.3333, A 0.000, B 0.000, C 0.000 }
gfCNCPoint5[745] = {X 250.8349, Y 7.8699, Z -6.3333, A 0.000, B 0.000, C 0.000 }
gfCNCPoint5[746] = {X 266.7633, Y 7.8699, Z -6.3333, A 0.000, B 0.000, C 0.000 }
gfCNCPoint5[747] = {X 267.7186, Y 7.9847, Z -6.3333, A 0.000, B 0.000, C 0.000 }
gfCNCPoint5[748] = {X 268.6249, Y 8.3079, Z -6.3333, A 0.000, B 0.000, C 0.000 }
gfCNCPoint5[749] = {X 269.4372, Y 8.8236, Z -6.3333, A 0.000, B 0.000, C 0.000 }
gfCNCPoint5[750] = {X 270.1152, Y 9.5063, Z -6.3333, A 0.000, B 0.000, C 0.000 }
gfCNCPoint5[751] = {X 270.6255, Y 10.3220, Z -6.3333, A 0.000, B 0.000, C 0.000 }
gfCNCPoint5[752] = {X 270.9427, Y 11.2304, Z -6.3333, A 0.000, B 0.000, C 0.000 }
gfCNCPoint5[753] = {X 271.0510, Y 12.1864, Z -6.3333, A 0.000, B 0.000, C 0.000 }
gfCNCPoint5[754] = {X 271.0508, Y 13.0225, Z -6.3333, A 0.000, B 0.000, C 0.000 }
gfCNCPoint5[755] = {X 270.9425, Y 13.9402, Z -6.3333, A 0.000, B 0.000, C 0.000 }
gfCNCPoint5[756] = {X 270.6415, Y 14.8139, Z -6.3333, A 0.000, B 0.000, C 0.000 }
gfCNCPoint5[757] = {X 270.1616, Y 15.6036, Z -6.3333, A 0.000, B 0.000, C 0.000 }
gfCNCPoint5[758] = {X 269.5246, Y 16.2732, Z -6.3333, A 0.000, B 0.000, C 0.000 }
gfCNCPoint5[759] = {X 269.5245, Y 28.5936, Z -6.3333, A 0.000, B 0.000, C 0.000 }
gfCNCPoint5[760] = {X 273.5245, Y 28.5936, Z -6.3333, A 0.000, B 0.000, C 0.000 }
gfCNCPoint5[761] = {X 269.4445, Y 28.5936, Z -6.3333, A 0.000, B 0.000, C 0.000 }
gfCNCPoint5[762] = {X 269.4445, Y 40.9518, Z -6.3333, A 0.000, B 0.000, C 0.000 }
gfCNCPoint5[763] = {X 269.4866, Y 40.9863, Z -6.3333, A 0.000, B 0.000, C 0.000 }
gfCNCPoint5[764] = {X 270.1068, Y 41.6433, Z -6.3333, A 0.000, B 0.000, C 0.000 }
gfCNCPoint5[765] = {X 270.5738, Y 42.4169, Z -6.3333, A 0.000, B 0.000, C 0.000 }
gfCNCPoint5[766] = {X 270.8662, Y 43.2718, Z -6.3333, A 0.000, B 0.000, C 0.000 }
gfCNCPoint5[767] = {X 270.9708, Y 44.1693, Z -6.3333, A 0.000, B 0.000, C 0.000 }
gfCNCPoint5[768] = {X 270.9710, Y 45.0000, Z -6.3333, A 0.000, B 0.000, C 0.000 }
gfCNCPoint5[769] = {X 270.8647, Y 45.9435, Z -6.3333, A 0.000, B 0.000, C 0.000 }
gfCNCPoint5[770] = {X 270.5511, Y 46.8397, Z -6.3333, A 0.000, B 0.000, C 0.000 }
gfCNCPoint5[771] = {X 270.0460, Y 47.6436, Z -6.3333, A 0.000, B 0.000, C 0.000 }
gfCNCPoint5[772] = {X 269.3746, Y 48.3150, Z -6.3333, A 0.000, B 0.000, C 0.000 }
gfCNCPoint5[773] = {X 268.5707, Y 48.8201, Z -6.3333, A 0.000, B 0.000, C 0.000 }
gfCNCPoint5[774] = {X 267.6745, Y 49.1337, Z -6.3333, A 0.000, B 0.000, C 0.000 }
gfCNCPoint5[775] = {X 266.7310, Y 49.2400, Z -6.3333, A 0.000, B 0.000, C 0.000 }
gfCNCPoint5[776] = {X 260.2876, Y 49.2400, Z -6.3333, A 0.000, B 0.000, C 0.000 }
gfCNCPoint5[777] = {X 259.3487, Y 49.1347, Z -6.3333, A 0.000, B 0.000, C 0.000 }
gfCNCPoint5[778] = {X 258.4564, Y 48.8242, Z -6.3333, A 0.000, B 0.000, C 0.000 }
gfCNCPoint5[779] = {X 257.6550, Y 48.3238, Z -6.3333, A 0.000, B 0.000, C 0.000 }
gfCNCPoint5[780] = {X 256.9844, Y 47.6583, Z -6.3333, A 0.000, B 0.000, C 0.000 }
gfCNCPoint5[781] = {X 256.4777, Y 46.8609, Z -6.3333, A 0.000, B 0.000, C 0.000 }
gfCNCPoint5[782] = {X 256.1603, Y 45.9711, Z -6.3333, A 0.000, B 0.000, C 0.000 }
gfCNCPoint5[783] = {X 256.0477, Y 45.0330, Z -6.3333, A 0.000, B 0.000, C 0.000 }
gfCNCPoint5[784] = {X 256.0480, Y 44.1505, Z -6.3333, A 0.000, B 0.000, C 0.000 }
gfCNCPoint5[785] = {X 256.1585, Y 43.2454, Z -6.3333, A 0.000, B 0.000, C 0.000 }
gfCNCPoint5[786] = {X 256.4599, Y 42.3850, Z -6.3333, A 0.000, B 0.000, C 0.000 }
gfCNCPoint5[787] = {X 256.9383, Y 41.6088, Z -6.3333, A 0.000, B 0.000, C 0.000 }
gfCNCPoint5[788] = {X 257.5715, Y 40.9529, Z -6.3333, A 0.000, B 0.000, C 0.000 }
gfCNCPoint5[789] = {X 257.5715, Y 34.3938, Z -6.3333, A 0.000, B 0.000, C 0.000 }
gfCNCPoint5[790] = {X 254.7195, Y 34.3938, Z -6.3333, A 0.000, B 0.000, C 0.000 }
gfCNCPoint5[791] = {X 250.3972, Y 42.8128, Z -6.3333, A 0.000, B 0.000, C 0.000 }
gfCNCPoint5[792] = {X 250.5710, Y 43.4832, Z -6.3333, A 0.000, B 0.000, C 0.000 }
gfCNCPoint5[793] = {X 250.6334, Y 44.1730, Z -6.3333, A 0.000, B 0.000, C 0.000 }
gfCNCPoint5[794] = {X 250.6336, Y 45.0000, Z -6.3333, A 0.000, B 0.000, C 0.000 }
gfCNCPoint5[795] = {X 250.5273, Y 45.9435, Z -6.3333, A 0.000, B 0.000, C 0.000 }
gfCNCPoint5[796] = {X 250.2137, Y 46.8397, Z -6.3333, A 0.000, B 0.000, C 0.000 }
gfCNCPoint5[797] = {X 249.7085, Y 47.6436, Z -6.3333, A 0.000, B 0.000, C 0.000 }
gfCNCPoint5[798] = {X 249.0372, Y 48.3150, Z -6.3333, A 0.000, B 0.000, C 0.000 }
gfCNCPoint5[799] = {X 248.2332, Y 48.8201, Z -6.3333, A 0.000, B 0.000, C 0.000 }
gfCNCPoint5[800] = {X 247.3370, Y 49.1337, Z -6.3333, A 0.000, B 0.000, C 0.000 }
gfCNCPoint5[801] = {X 246.3936, Y 49.2400, Z -6.3333, A 0.000, B 0.000, C 0.000 }
gfCNCPoint5[802] = {X 239.8075, Y 49.2400, Z -6.3333, A 0.000, B 0.000, C 0.000 }
gfCNCPoint5[803] = {X 238.8640, Y 49.1337, Z -6.3333, A 0.000, B 0.000, C 0.000 }
gfCNCPoint5[804] = {X 237.9679, Y 48.8201, Z -6.3333, A 0.000, B 0.000, C 0.000 }
gfCNCPoint5[805] = {X 237.1639, Y 48.3150, Z -6.3333, A 0.000, B 0.000, C 0.000 }
gfCNCPoint5[806] = {X 236.4926, Y 47.6436, Z -6.3333, A 0.000, B 0.000, C 0.000 }
gfCNCPoint5[807] = {X 235.9874, Y 46.8397, Z -6.3333, A 0.000, B 0.000, C 0.000 }
gfCNCPoint5[808] = {X 235.6738, Y 45.9436, Z -6.3333, A 0.000, B 0.000, C 0.000 }
gfCNCPoint5[809] = {X 235.5675, Y 45.0001, Z -6.3333, A 0.000, B 0.000, C 0.000 }
gfCNCPoint5[810] = {X 235.5679, Y 44.1505, Z -6.3333, A 0.000, B 0.000, C 0.000 }
gfCNCPoint5[811] = {X 235.6649, Y 43.3054, Z -6.3333, A 0.000, B 0.000, C 0.000 }
gfCNCPoint5[812] = {X 235.9285, Y 42.4967, Z -6.3333, A 0.000, B 0.000, C 0.000 }
gfCNCPoint5[813] = {X 236.3483, Y 41.7570, Z -6.3333, A 0.000, B 0.000, C 0.000 }
gfCNCPoint5[814] = {X 236.9073, Y 41.1158, Z -6.3333, A 0.000, B 0.000, C 0.000 }
gfCNCPoint5[815] = {X 237.5830, Y 40.5992, Z -6.3333, A 0.000, B 0.000, C 0.000 }
gfCNCPoint5[816] = {X 238.3482, Y 40.2278, Z -6.3333, A 0.000, B 0.000, C 0.000 }
gfCNCPoint5[817] = {X 242.3857, Y 32.3248, Z -6.3333, A 0.000, B 0.000, C 0.000 }
gfCNCPoint5[818] = {X 241.2087, Y 31.5440, Z -6.3333, A 0.000, B 0.000, C 0.000 }
gfCNCPoint5[819] = {X 240.1389, Y 30.6218, Z -6.3333, A 0.000, B 0.000, C 0.000 }
gfCNCPoint5[820] = {X 239.1931, Y 29.5728, Z -6.3333, A 0.000, B 0.000, C 0.000 }
gfCNCPoint5[821] = {X 238.3864, Y 28.4134, Z -6.3333, A 0.000, B 0.000, C 0.000 }
gfCNCPoint5[822] = {X 237.7314, Y 27.1620, Z -6.3333, A 0.000, B 0.000, C 0.000 }
gfCNCPoint5[823] = {X 237.2385, Y 25.8383, Z -6.3333, A 0.000, B 0.000, C 0.000 }
gfCNCPoint5[824] = {X 236.8205, Y 24.0358, Z -6.3333, A 0.000, B 0.000, C 0.000 }
gfCNCPoint5[825] = {X 236.6075, Y 22.1976, Z -6.3333, A 0.000, B 0.000, C 0.000 }
gfCNCPoint5[826] = {X 236.6022, Y 20.3472, Z -6.3333, A 0.000, B 0.000, C 0.000 }
gfCNCPoint5[827] = {X 236.8047, Y 18.5079, Z -6.3333, A 0.000, B 0.000, C 0.000 }
gfCNCPoint5[828] = {X 237.2124, Y 16.7030, Z -6.3333, A 0.000, B 0.000, C 0.000 }
gfCNCPoint5[829] = {X 237.7790, Y 15.1378, Z -6.3333, A 0.000, B 0.000, C 0.000 }
gfCNCPoint5[830] = {X 238.5608, Y 13.6681, Z -6.3333, A 0.000, B 0.000, C 0.000 }
gfCNCPoint5[831] = {X 239.5421, Y 12.3235, Z -6.3333, A 0.000, B 0.000, C 0.000 }
gfCNCPoint5[832] = {X 240.7033, Y 11.1308, Z -6.3333, A 0.000, B 0.000, C 0.000 }
gfCNCPoint5[833] = {X 242.0212, Y 10.1138, Z -6.3333, A 0.000, B 0.000, C 0.000 }
gfCNCPoint5[834] = {X 243.4693, Y 9.2929, Z -6.3333, A 0.000, B 0.000, C 0.000 }
gfCNCPoint5[835] = {X 245.0188, Y 8.6845, Z -6.3333, A 0.000, B 0.000, C 0.000 }
gfCNCPoint5[836] = {X 246.6386, Y 8.3008, Z -6.3333, A 0.000, B 0.000, C 0.000 }
gfCNCPoint5[837] = {X 248.7286, Y 8.0302, Z -6.3333, A 0.000, B 0.000, C 0.000 }
gfCNCPoint5[838] = {X 250.8346, Y 7.9499, Z -6.3333, A 0.000, B 0.000, C 0.000 }
gfCNCPoint5[839] = {X 266.7627, Y 7.9499, Z -6.3333, A 0.000, B 0.000, C 0.000 }
gfCNCPoint5[840] = {X 267.7003, Y 8.0626, Z -6.3333, A 0.000, B 0.000, C 0.000 }
gfCNCPoint5[841] = {X 268.5898, Y 8.3798, Z -6.3333, A 0.000, B 0.000, C 0.000 }
gfCNCPoint5[842] = {X 269.3870, Y 8.8860, Z -6.3333, A 0.000, B 0.000, C 0.000 }
gfCNCPoint5[843] = {X 270.0526, Y 9.5560, Z -6.3333, A 0.000, B 0.000, C 0.000 }
gfCNCPoint5[844] = {X 270.5534, Y 10.3566, Z -6.3333, A 0.000, B 0.000, C 0.000 }
gfCNCPoint5[845] = {X 270.8647, Y 11.2482, Z -6.3333, A 0.000, B 0.000, C 0.000 }
gfCNCPoint5[846] = {X 270.9710, Y 12.1865, Z -6.3333, A 0.000, B 0.000, C 0.000 }
gfCNCPoint5[847] = {X 270.9708, Y 13.0217, Z -6.3333, A 0.000, B 0.000, C 0.000 }
gfCNCPoint5[848] = {X 270.8625, Y 13.9314, Z -6.3333, A 0.000, B 0.000, C 0.000 }
gfCNCPoint5[849] = {X 270.5612, Y 14.7966, Z -6.3333, A 0.000, B 0.000, C 0.000 }
gfCNCPoint5[850] = {X 270.0811, Y 15.5770, Z -6.3333, A 0.000, B 0.000, C 0.000 }
gfCNCPoint5[851] = {X 269.4446, Y 16.2359, Z -6.3333, A 0.000, B 0.000, C 0.000 }
gfCNCPoint5[852] = {X 269.4445, Y 28.5936, Z -6.3333, A 0.000, B 0.000, C 0.000 }
gfCNCPoint5[853] = {X 273.4445, Y 28.5936, Z -6.3333, A 0.000, B 0.000, C 0.000 }
gfCNCPoint5[854] = {X 269.3645, Y 28.5935, Z -6.3333, A 0.000, B 0.000, C 0.000 }
gfCNCPoint5[855] = {X 269.3645, Y 40.9897, Z -6.3333, A 0.000, B 0.000, C 0.000 }
gfCNCPoint5[856] = {X 269.4352, Y 41.0476, Z -6.3333, A 0.000, B 0.000, C 0.000 }
gfCNCPoint5[857] = {X 270.0435, Y 41.6922, Z -6.3333, A 0.000, B 0.000, C 0.000 }
gfCNCPoint5[858] = {X 270.5014, Y 42.4511, Z -6.3333, A 0.000, B 0.000, C 0.000 }
gfCNCPoint5[859] = {X 270.7882, Y 43.2897, Z -6.3333, A 0.000, B 0.000, C 0.000 }
gfCNCPoint5[860] = {X 270.8909, Y 44.1700, Z -6.3333, A 0.000, B 0.000, C 0.000 }
gfCNCPoint5[861] = {X 270.8910, Y 45.0000, Z -6.3333, A 0.000, B 0.000, C 0.000 }
gfCNCPoint5[862] = {X 270.7867, Y 45.9257, Z -6.3333, A 0.000, B 0.000, C 0.000 }
gfCNCPoint5[863] = {X 270.4791, Y 46.8050, Z -6.3333, A 0.000, B 0.000, C 0.000 }
gfCNCPoint5[864] = {X 269.9835, Y 47.5937, Z -6.3333, A 0.000, B 0.000, C 0.000 }
gfCNCPoint5[865] = {X 269.3247, Y 48.2524, Z -6.3333, A 0.000, B 0.000, C 0.000 }
gfCNCPoint5[866] = {X 268.5360, Y 48.7480, Z -6.3333, A 0.000, B 0.000, C 0.000 }
gfCNCPoint5[867] = {X 267.6567, Y 49.0557, Z -6.3333, A 0.000, B 0.000, C 0.000 }
gfCNCPoint5[868] = {X 266.7310, Y 49.1600, Z -6.3333, A 0.000, B 0.000, C 0.000 }
gfCNCPoint5[869] = {X 260.2876, Y 49.1600, Z -6.3333, A 0.000, B 0.000, C 0.000 }
gfCNCPoint5[870] = {X 259.3664, Y 49.0567, Z -6.3333, A 0.000, B 0.000, C 0.000 }
gfCNCPoint5[871] = {X 258.4910, Y 48.7520, Z -6.3333, A 0.000, B 0.000, C 0.000 }
gfCNCPoint5[872] = {X 257.7047, Y 48.2611, Z -6.3333, A 0.000, B 0.000, C 0.000 }
gfCNCPoint5[873] = {X 257.0467, Y 47.6082, Z -6.3333, A 0.000, B 0.000, C 0.000 }
gfCNCPoint5[874] = {X 256.5496, Y 46.8258, Z -6.3333, A 0.000, B 0.000, C 0.000 }
gfCNCPoint5[875] = {X 256.2381, Y 45.9527, Z -6.3333, A 0.000, B 0.000, C 0.000 }
gfCNCPoint5[876] = {X 256.1277, Y 45.0324, Z -6.3333, A 0.000, B 0.000, C 0.000 }
gfCNCPoint5[877] = {X 256.1280, Y 44.1516, Z -6.3333, A 0.000, B 0.000, C 0.000 }
gfCNCPoint5[878] = {X 256.2385, Y 43.2545, Z -6.3333, A 0.000, B 0.000, C 0.000 }
gfCNCPoint5[879] = {X 256.5401, Y 42.4026, Z -6.3333, A 0.000, B 0.000, C 0.000 }
gfCNCPoint5[880] = {X 257.0187, Y 41.6358, Z -6.3333, A 0.000, B 0.000, C 0.000 }
gfCNCPoint5[881] = {X 257.6515, Y 40.9906, Z -6.3333, A 0.000, B 0.000, C 0.000 }
gfCNCPoint5[882] = {X 257.6515, Y 34.3138, Z -6.3333, A 0.000, B 0.000, C 0.000 }
gfCNCPoint5[883] = {X 254.6706, Y 34.3138, Z -6.3333, A 0.000, B 0.000, C 0.000 }
gfCNCPoint5[884] = {X 250.3103, Y 42.8070, Z -6.3333, A 0.000, B 0.000, C 0.000 }
gfCNCPoint5[885] = {X 250.4892, Y 43.4801, Z -6.3333, A 0.000, B 0.000, C 0.000 }
gfCNCPoint5[886] = {X 250.5534, Y 44.1736, Z -6.3333, A 0.000, B 0.000, C 0.000 }
gfCNCPoint5[887] = {X 250.5536, Y 45.0000, Z -6.3333, A 0.000, B 0.000, C 0.000 }
gfCNCPoint5[888] = {X 250.4493, Y 45.9257, Z -6.3333, A 0.000, B 0.000, C 0.000 }
gfCNCPoint5[889] = {X 250.1416, Y 46.8050, Z -6.3333, A 0.000, B 0.000, C 0.000 }
gfCNCPoint5[890] = {X 249.6460, Y 47.5937, Z -6.3333, A 0.000, B 0.000, C 0.000 }
gfCNCPoint5[891] = {X 248.9873, Y 48.2524, Z -6.3333, A 0.000, B 0.000, C 0.000 }
gfCNCPoint5[892] = {X 248.1985, Y 48.7480, Z -6.3333, A 0.000, B 0.000, C 0.000 }
gfCNCPoint5[893] = {X 247.3192, Y 49.0557, Z -6.3333, A 0.000, B 0.000, C 0.000 }
gfCNCPoint5[894] = {X 246.3936, Y 49.1600, Z -6.3333, A 0.000, B 0.000, C 0.000 }
gfCNCPoint5[895] = {X 239.8075, Y 49.1600, Z -6.3333, A 0.000, B 0.000, C 0.000 }
gfCNCPoint5[896] = {X 238.8818, Y 49.0557, Z -6.3333, A 0.000, B 0.000, C 0.000 }
gfCNCPoint5[897] = {X 238.0026, Y 48.7480, Z -6.3333, A 0.000, B 0.000, C 0.000 }
gfCNCPoint5[898] = {X 237.2138, Y 48.2524, Z -6.3333, A 0.000, B 0.000, C 0.000 }
gfCNCPoint5[899] = {X 236.5551, Y 47.5937, Z -6.3333, A 0.000, B 0.000, C 0.000 }
gfCNCPoint5[900] = {X 236.0595, Y 46.8050, Z -6.3333, A 0.000, B 0.000, C 0.000 }
gfCNCPoint5[901] = {X 235.7518, Y 45.9257, Z -6.3333, A 0.000, B 0.000, C 0.000 }
gfCNCPoint5[902] = {X 235.6475, Y 45.0000, Z -6.3333, A 0.000, B 0.000, C 0.000 }
gfCNCPoint5[903] = {X 235.6479, Y 44.1516, Z -6.3333, A 0.000, B 0.000, C 0.000 }
gfCNCPoint5[904] = {X 235.7441, Y 43.3174, Z -6.3333, A 0.000, B 0.000, C 0.000 }
gfCNCPoint5[905] = {X 236.0059, Y 42.5195, Z -6.3333, A 0.000, B 0.000, C 0.000 }
gfCNCPoint5[906] = {X 236.4226, Y 41.7905, Z -6.3333, A 0.000, B 0.000, C 0.000 }
gfCNCPoint5[907] = {X 236.9772, Y 41.1600, Z -6.3333, A 0.000, B 0.000, C 0.000 }
gfCNCPoint5[908] = {X 237.6471, Y 40.6537, Z -6.3333, A 0.000, B 0.000, C 0.000 }
gfCNCPoint5[909] = {X 238.4051, Y 40.2923, Z -6.3333, A 0.000, B 0.000, C 0.000 }
gfCNCPoint5[910] = {X 242.4917, Y 32.2932, Z -6.3333, A 0.000, B 0.000, C 0.000 }
gfCNCPoint5[911] = {X 241.3076, Y 31.5184, Z -6.3333, A 0.000, B 0.000, C 0.000 }
gfCNCPoint5[912] = {X 240.2311, Y 30.6000, Z -6.3333, A 0.000, B 0.000, C 0.000 }
gfCNCPoint5[913] = {X 239.2794, Y 29.5528, Z -6.3333, A 0.000, B 0.000, C 0.000 }
gfCNCPoint5[914] = {X 238.4679, Y 28.3936, Z -6.3333, A 0.000, B 0.000, C 0.000 }
gfCNCPoint5[915] = {X 237.8096, Y 27.1410, Z -6.3333, A 0.000, B 0.000, C 0.000 }
gfCNCPoint5[916] = {X 237.3151, Y 25.8152, Z -6.3333, A 0.000, B 0.000, C 0.000 }
gfCNCPoint5[917] = {X 236.8992, Y 24.0215, Z -6.3333, A 0.000, B 0.000, C 0.000 }
gfCNCPoint5[918] = {X 236.6873, Y 22.1924, Z -6.3333, A 0.000, B 0.000, C 0.000 }
gfCNCPoint5[919] = {X 236.6821, Y 20.3511, Z -6.3333, A 0.000, B 0.000, C 0.000 }
gfCNCPoint5[920] = {X 236.8836, Y 18.5209, Z -6.3333, A 0.000, B 0.000, C 0.000 }
gfCNCPoint5[921] = {X 237.2893, Y 16.7249, Z -6.3333, A 0.000, B 0.000, C 0.000 }
gfCNCPoint5[922] = {X 237.8522, Y 15.1702, Z -6.3333, A 0.000, B 0.000, C 0.000 }
gfCNCPoint5[923] = {X 238.6287, Y 13.7105, Z -6.3333, A 0.000, B 0.000, C 0.000 }
gfCNCPoint5[924] = {X 239.6034, Y 12.3750, Z -6.3333, A 0.000, B 0.000, C 0.000 }
gfCNCPoint5[925] = {X 240.7567, Y 11.1903, Z -6.3333, A 0.000, B 0.000, C 0.000 }
gfCNCPoint5[926] = {X 242.0657, Y 10.1802, Z -6.3333, A 0.000, B 0.000, C 0.000 }
gfCNCPoint5[927] = {X 243.5041, Y 9.3649, Z -6.3333, A 0.000, B 0.000, C 0.000 }
gfCNCPoint5[928] = {X 245.0431, Y 8.7607, Z -6.3333, A 0.000, B 0.000, C 0.000 }
gfCNCPoint5[929] = {X 246.6520, Y 8.3797, Z -6.3333, A 0.000, B 0.000, C 0.000 }
gfCNCPoint5[930] = {X 248.7352, Y 8.1099, Z -6.3333, A 0.000, B 0.000, C 0.000 }
gfCNCPoint5[931] = {X 250.8343, Y 8.0299, Z -6.3333, A 0.000, B 0.000, C 0.000 }
gfCNCPoint5[932] = {X 266.7621, Y 8.0299, Z -6.3333, A 0.000, B 0.000, C 0.000 }
gfCNCPoint5[933] = {X 267.6820, Y 8.1404, Z -6.3333, A 0.000, B 0.000, C 0.000 }
gfCNCPoint5[934] = {X 268.5547, Y 8.4517, Z -6.3333, A 0.000, B 0.000, C 0.000 }
gfCNCPoint5[935] = {X 269.3369, Y 8.9483, Z -6.3333, A 0.000, B 0.000, C 0.000 }
gfCNCPoint5[936] = {X 269.9899, Y 9.6057, Z -6.3333, A 0.000, B 0.000, C 0.000 }
gfCNCPoint5[937] = {X 270.4812, Y 10.3912, Z -6.3333, A 0.000, B 0.000, C 0.000 }
gfCNCPoint5[938] = {X 270.7867, Y 11.2660, Z -6.3333, A 0.000, B 0.000, C 0.000 }
gfCNCPoint5[939] = {X 270.8910, Y 12.1866, Z -6.3333, A 0.000, B 0.000, C 0.000 }
gfCNCPoint5[940] = {X 270.8908, Y 13.0208, Z -6.3333, A 0.000, B 0.000, C 0.000 }
gfCNCPoint5[941] = {X 270.7824, Y 13.9225, Z -6.3333, A 0.000, B 0.000, C 0.000 }
gfCNCPoint5[942] = {X 270.4809, Y 14.7792, Z -6.3333, A 0.000, B 0.000, C 0.000 }
gfCNCPoint5[943] = {X 270.0007, Y 15.5500, Z -6.3333, A 0.000, B 0.000, C 0.000 }
gfCNCPoint5[944] = {X 269.3646, Y 16.1982, Z -6.3333, A 0.000, B 0.000, C 0.000 }
gfCNCPoint5[945] = {X 269.3645, Y 28.5935, Z -6.3333, A 0.000, B 0.000, C 0.000 }
gfCNCPoint5[946] = {X 273.3645, Y 28.5936, Z -6.3333, A 0.000, B 0.000, C 0.000 }
gfCNCPoint5[947] = {X 269.2845, Y 28.5935, Z -6.3333, A 0.000, B 0.000, C 0.000 }
gfCNCPoint5[948] = {X 269.2845, Y 41.0276, Z -6.3333, A 0.000, B 0.000, C 0.000 }
gfCNCPoint5[949] = {X 269.3839, Y 41.1090, Z -6.3333, A 0.000, B 0.000, C 0.000 }
gfCNCPoint5[950] = {X 269.9802, Y 41.7411, Z -6.3333, A 0.000, B 0.000, C 0.000 }
gfCNCPoint5[951] = {X 270.4291, Y 42.4853, Z -6.3333, A 0.000, B 0.000, C 0.000 }
gfCNCPoint5[952] = {X 270.7103, Y 43.3076, Z -6.3333, A 0.000, B 0.000, C 0.000 }
gfCNCPoint5[953] = {X 270.8109, Y 44.1708, Z -6.3333, A 0.000, B 0.000, C 0.000 }
gfCNCPoint5[954] = {X 270.8110, Y 45.0000, Z -6.3333, A 0.000, B 0.000, C 0.000 }
gfCNCPoint5[955] = {X 270.7087, Y 45.9079, Z -6.3333, A 0.000, B 0.000, C 0.000 }
gfCNCPoint5[956] = {X 270.4070, Y 46.7702, Z -6.3333, A 0.000, B 0.000, C 0.000 }
gfCNCPoint5[957] = {X 269.9209, Y 47.5438, Z -6.3333, A 0.000, B 0.000, C 0.000 }
gfCNCPoint5[958] = {X 269.2749, Y 48.1899, Z -6.3333, A 0.000, B 0.000, C 0.000 }
gfCNCPoint5[959] = {X 268.5013, Y 48.6760, Z -6.3333, A 0.000, B 0.000, C 0.000 }
gfCNCPoint5[960] = {X 267.6389, Y 48.9777, Z -6.3333, A 0.000, B 0.000, C 0.000 }
gfCNCPoint5[961] = {X 266.7310, Y 49.0800, Z -6.3333, A 0.000, B 0.000, C 0.000 }
gfCNCPoint5[962] = {X 260.2876, Y 49.0800, Z -6.3333, A 0.000, B 0.000, C 0.000 }
gfCNCPoint5[963] = {X 259.3841, Y 48.9787, Z -6.3333, A 0.000, B 0.000, C 0.000 }
gfCNCPoint5[964] = {X 258.5255, Y 48.6799, Z -6.3333, A 0.000, B 0.000, C 0.000 }
gfCNCPoint5[965] = {X 257.7544, Y 48.1983, Z -6.3333, A 0.000, B 0.000, C 0.000 }
gfCNCPoint5[966] = {X 257.1090, Y 47.5580, Z -6.3333, A 0.000, B 0.000, C 0.000 }
gfCNCPoint5[967] = {X 256.6215, Y 46.7907, Z -6.3333, A 0.000, B 0.000, C 0.000 }
gfCNCPoint5[968] = {X 256.3160, Y 45.9344, Z -6.3333, A 0.000, B 0.000, C 0.000 }
gfCNCPoint5[969] = {X 256.2077, Y 45.0318, Z -6.3333, A 0.000, B 0.000, C 0.000 }
gfCNCPoint5[970] = {X 256.2080, Y 44.1527, Z -6.3333, A 0.000, B 0.000, C 0.000 }
gfCNCPoint5[971] = {X 256.3185, Y 43.2637, Z -6.3333, A 0.000, B 0.000, C 0.000 }
gfCNCPoint5[972] = {X 256.6204, Y 42.4203, Z -6.3333, A 0.000, B 0.000, C 0.000 }
gfCNCPoint5[973] = {X 257.0991, Y 41.6631, Z -6.3333, A 0.000, B 0.000, C 0.000 }
gfCNCPoint5[974] = {X 257.7315, Y 41.0287, Z -6.3333, A 0.000, B 0.000, C 0.000 }
gfCNCPoint5[975] = {X 257.7315, Y 34.2338, Z -6.3333, A 0.000, B 0.000, C 0.000 }
gfCNCPoint5[976] = {X 254.6218, Y 34.2338, Z -6.3333, A 0.000, B 0.000, C 0.000 }
gfCNCPoint5[977] = {X 250.2232, Y 42.8015, Z -6.3333, A 0.000, B 0.000, C 0.000 }
gfCNCPoint5[978] = {X 250.4074, Y 43.4771, Z -6.3333, A 0.000, B 0.000, C 0.000 }
gfCNCPoint5[979] = {X 250.4734, Y 44.1743, Z -6.3333, A 0.000, B 0.000, C 0.000 }
gfCNCPoint5[980] = {X 250.4736, Y 45.0000, Z -6.3333, A 0.000, B 0.000, C 0.000 }
gfCNCPoint5[981] = {X 250.3713, Y 45.9079, Z -6.3333, A 0.000, B 0.000, C 0.000 }
gfCNCPoint5[982] = {X 250.0695, Y 46.7702, Z -6.3333, A 0.000, B 0.000, C 0.000 }
gfCNCPoint5[983] = {X 249.5834, Y 47.5438, Z -6.3333, A 0.000, B 0.000, C 0.000 }
gfCNCPoint5[984] = {X 248.9374, Y 48.1899, Z -6.3333, A 0.000, B 0.000, C 0.000 }
gfCNCPoint5[985] = {X 248.1638, Y 48.6760, Z -6.3333, A 0.000, B 0.000, C 0.000 }
gfCNCPoint5[986] = {X 247.3014, Y 48.9777, Z -6.3333, A 0.000, B 0.000, C 0.000 }
gfCNCPoint5[987] = {X 246.3936, Y 49.0800, Z -6.3333, A 0.000, B 0.000, C 0.000 }
gfCNCPoint5[988] = {X 239.8075, Y 49.0800, Z -6.3333, A 0.000, B 0.000, C 0.000 }
gfCNCPoint5[989] = {X 238.8996, Y 48.9777, Z -6.3333, A 0.000, B 0.000, C 0.000 }
gfCNCPoint5[990] = {X 238.0373, Y 48.6760, Z -6.3333, A 0.000, B 0.000, C 0.000 }
gfCNCPoint5[991] = {X 237.2637, Y 48.1899, Z -6.3333, A 0.000, B 0.000, C 0.000 }
gfCNCPoint5[992] = {X 236.6176, Y 47.5438, Z -6.3333, A 0.000, B 0.000, C 0.000 }
gfCNCPoint5[993] = {X 236.1315, Y 46.7702, Z -6.3333, A 0.000, B 0.000, C 0.000 }
gfCNCPoint5[994] = {X 235.8298, Y 45.9079, Z -6.3333, A 0.000, B 0.000, C 0.000 }
gfCNCPoint5[995] = {X 235.7275, Y 45.0000, Z -6.3333, A 0.000, B 0.000, C 0.000 }
gfCNCPoint5[996] = {X 235.7279, Y 44.1527, Z -6.3333, A 0.000, B 0.000, C 0.000 }
gfCNCPoint5[997] = {X 235.8234, Y 43.3294, Z -6.3333, A 0.000, B 0.000, C 0.000 }
gfCNCPoint5[998] = {X 236.0833, Y 42.5424, Z -6.3333, A 0.000, B 0.000, C 0.000 }
gfCNCPoint5[999] = {X 236.4969, Y 41.8242, Z -6.3333, A 0.000, B 0.000, C 0.000 }
gfCNCPoint5[1000] = {X 237.0471, Y 41.2044, Z -6.3333, A 0.000, B 0.000, C 0.000 }
gfCNCPoint5[1001] = {X 237.7112, Y 40.7085, Z -6.3333, A 0.000, B 0.000, C 0.000 }
gfCNCPoint5[1002] = {X 238.4618, Y 40.3571, Z -6.3333, A 0.000, B 0.000, C 0.000 }
gfCNCPoint5[1003] = {X 242.5979, Y 32.2612, Z -6.3333, A 0.000, B 0.000, C 0.000 }
gfCNCPoint5[1004] = {X 241.4068, Y 31.4925, Z -6.3333, A 0.000, B 0.000, C 0.000 }
gfCNCPoint5[1005] = {X 240.3235, Y 30.5780, Z -6.3333, A 0.000, B 0.000, C 0.000 }
gfCNCPoint5[1006] = {X 239.3659, Y 29.5327, Z -6.3333, A 0.000, B 0.000, C 0.000 }
gfCNCPoint5[1007] = {X 238.5496, Y 28.3737, Z -6.3333, A 0.000, B 0.000, C 0.000 }
gfCNCPoint5[1008] = {X 237.8879, Y 27.1200, Z -6.3333, A 0.000, B 0.000, C 0.000 }
gfCNCPoint5[1009] = {X 237.3917, Y 25.7920, Z -6.3333, A 0.000, B 0.000, C 0.000 }
gfCNCPoint5[1010] = {X 236.9779, Y 24.0072, Z -6.3333, A 0.000, B 0.000, C 0.000 }
gfCNCPoint5[1011] = {X 236.7671, Y 22.1872, Z -6.3333, A 0.000, B 0.000, C 0.000 }
gfCNCPoint5[1012] = {X 236.7620, Y 20.3551, Z -6.3333, A 0.000, B 0.000, C 0.000 }
gfCNCPoint5[1013] = {X 236.9625, Y 18.5340, Z -6.3333, A 0.000, B 0.000, C 0.000 }
gfCNCPoint5[1014] = {X 237.3663, Y 16.7469, Z -6.3333, A 0.000, B 0.000, C 0.000 }
gfCNCPoint5[1015] = {X 237.9252, Y 15.2028, Z -6.3333, A 0.000, B 0.000, C 0.000 }
gfCNCPoint5[1016] = {X 238.6965, Y 13.7530, Z -6.3333, A 0.000, B 0.000, C 0.000 }
gfCNCPoint5[1017] = {X 239.6645, Y 12.4265, Z -6.3333, A 0.000, B 0.000, C 0.000 }
gfCNCPoint5[1018] = {X 240.8101, Y 11.2499, Z -6.3333, A 0.000, B 0.000, C 0.000 }
gfCNCPoint5[1019] = {X 242.1102, Y 10.2467, Z -6.3333, A 0.000, B 0.000, C 0.000 }
gfCNCPoint5[1020] = {X 243.5388, Y 9.4370, Z -6.3333, A 0.000, B 0.000, C 0.000 }
gfCNCPoint5[1021] = {X 245.0674, Y 8.8369, Z -6.3333, A 0.000, B 0.000, C 0.000 }
gfCNCPoint5[1022] = {X 246.6654, Y 8.4585, Z -6.3333, A 0.000, B 0.000, C 0.000 }
gfCNCPoint5[1023] = {X 248.7417, Y 8.1896, Z -6.3333, A 0.000, B 0.000, C 0.000 }
gfCNCPoint5[1024] = {X 250.8339, Y 8.1099, Z -6.3333, A 0.000, B 0.000, C 0.000 }
gfCNCPoint5[1025] = {X 266.7614, Y 8.1099, Z -6.3333, A 0.000, B 0.000, C 0.000 }
gfCNCPoint5[1026] = {X 267.6637, Y 8.2183, Z -6.3333, A 0.000, B 0.000, C 0.000 }
gfCNCPoint5[1027] = {X 268.5196, Y 8.5236, Z -6.3333, A 0.000, B 0.000, C 0.000 }
gfCNCPoint5[1028] = {X 269.2868, Y 9.0107, Z -6.3333, A 0.000, B 0.000, C 0.000 }
gfCNCPoint5[1029] = {X 269.9272, Y 9.6554, Z -6.3333, A 0.000, B 0.000, C 0.000 }
gfCNCPoint5[1030] = {X 270.4091, Y 10.4258, Z -6.3333, A 0.000, B 0.000, C 0.000 }
gfCNCPoint5[1031] = {X 270.7087, Y 11.2838, Z -6.3333, A 0.000, B 0.000, C 0.000 }
gfCNCPoint5[1032] = {X 270.8110, Y 12.1867, Z -6.3333, A 0.000, B 0.000, C 0.000 }
gfCNCPoint5[1033] = {X 270.8108, Y 13.0200, Z -6.3333, A 0.000, B 0.000, C 0.000 }
gfCNCPoint5[1034] = {X 270.7023, Y 13.9135, Z -6.3333, A 0.000, B 0.000, C 0.000 }
gfCNCPoint5[1035] = {X 270.4006, Y 14.7615, Z -6.3333, A 0.000, B 0.000, C 0.000 }
gfCNCPoint5[1036] = {X 269.9202, Y 15.5227, Z -6.3333, A 0.000, B 0.000, C 0.000 }
gfCNCPoint5[1037] = {X 269.2846, Y 16.1601, Z -6.3333, A 0.000, B 0.000, C 0.000 }
gfCNCPoint5[1038] = {X 269.2845, Y 28.5935, Z -6.3333, A 0.000, B 0.000, C 0.000 }
gfCNCPoint5[1039] = {X 273.2845, Y 28.5936, Z -6.3333, A 0.000, B 0.000, C 0.000 }
gfCNCPoint5[1040] = {X 269.2045, Y 28.5935, Z -6.3333, A 0.000, B 0.000, C 0.000 }
gfCNCPoint5[1041] = {X 269.2045, Y 41.0655, Z -6.3333, A 0.000, B 0.000, C 0.000 }
gfCNCPoint5[1042] = {X 269.3432, Y 41.1795, Z -6.3333, A 0.000, B 0.000, C 0.000 }
gfCNCPoint5[1043] = {X 269.9289, Y 41.8060, Z -6.3333, A 0.000, B 0.000, C 0.000 }
gfCNCPoint5[1044] = {X 270.3676, Y 42.5428, Z -6.3333, A 0.000, B 0.000, C 0.000 }
gfCNCPoint5[1045] = {X 270.6391, Y 43.3563, Z -6.3333, A 0.000, B 0.000, C 0.000 }
gfCNCPoint5[1046] = {X 270.7310, Y 44.2089, Z -6.3333, A 0.000, B 0.000, C 0.000 }
gfCNCPoint5[1047] = {X 270.7310, Y 45.0000, Z -6.3333, A 0.000, B 0.000, C 0.000 }
gfCNCPoint5[1048] = {X 270.6307, Y 45.8901, Z -6.3333, A 0.000, B 0.000, C 0.000 }
gfCNCPoint5[1049] = {X 270.3349, Y 46.7355, Z -6.3333, A 0.000, B 0.000, C 0.000 }
gfCNCPoint5[1050] = {X 269.8584, Y 47.4940, Z -6.3333, A 0.000, B 0.000, C 0.000 }
gfCNCPoint5[1051] = {X 269.2250, Y 48.1273, Z -6.3333, A 0.000, B 0.000, C 0.000 }
gfCNCPoint5[1052] = {X 268.4666, Y 48.6039, Z -6.3333, A 0.000, B 0.000, C 0.000 }
gfCNCPoint5[1053] = {X 267.6211, Y 48.8997, Z -6.3333, A 0.000, B 0.000, C 0.000 }
gfCNCPoint5[1054] = {X 266.7310, Y 49.0000, Z -6.3333, A 0.000, B 0.000, C 0.000 }
gfCNCPoint5[1055] = {X 260.2876, Y 49.0000, Z -6.3333, A 0.000, B 0.000, C 0.000 }
gfCNCPoint5[1056] = {X 259.3975, Y 48.8997, Z -6.3333, A 0.000, B 0.000, C 0.000 }
gfCNCPoint5[1057] = {X 258.5520, Y 48.6039, Z -6.3333, A 0.000, B 0.000, C 0.000 }
gfCNCPoint5[1058] = {X 257.7936, Y 48.1273, Z -6.3333, A 0.000, B 0.000, C 0.000 }
gfCNCPoint5[1059] = {X 257.1602, Y 47.4939, Z -6.3333, A 0.000, B 0.000, C 0.000 }
gfCNCPoint5[1060] = {X 256.6837, Y 46.7355, Z -6.3333, A 0.000, B 0.000, C 0.000 }
gfCNCPoint5[1061] = {X 256.3878, Y 45.8901, Z -6.3333, A 0.000, B 0.000, C 0.000 }
gfCNCPoint5[1062] = {X 256.2876, Y 45.0000, Z -6.3333, A 0.000, B 0.000, C 0.000 }
gfCNCPoint5[1063] = {X 256.2879, Y 44.1538, Z -6.3333, A 0.000, B 0.000, C 0.000 }
gfCNCPoint5[1064] = {X 256.3986, Y 43.2730, Z -6.3333, A 0.000, B 0.000, C 0.000 }
gfCNCPoint5[1065] = {X 256.7008, Y 42.4382, Z -6.3333, A 0.000, B 0.000, C 0.000 }
gfCNCPoint5[1066] = {X 257.1796, Y 41.6907, Z -6.3333, A 0.000, B 0.000, C 0.000 }
gfCNCPoint5[1067] = {X 257.8115, Y 41.0672, Z -6.3333, A 0.000, B 0.000, C 0.000 }
gfCNCPoint5[1068] = {X 257.8115, Y 34.1538, Z -6.3333, A 0.000, B 0.000, C 0.000 }
gfCNCPoint5[1069] = {X 254.8172, Y 34.1538, Z -6.3333, A 0.000, B 0.000, C 0.000 }
gfCNCPoint5[1070] = {X 254.5734, Y 34.1528, Z -6.3333, A 0.000, B 0.000, C 0.000 }
gfCNCPoint5[1071] = {X 250.1359, Y 42.7963, Z -6.3333, A 0.000, B 0.000, C 0.000 }
gfCNCPoint5[1072] = {X 250.3286, Y 43.4909, Z -6.3333, A 0.000, B 0.000, C 0.000 }
gfCNCPoint5[1073] = {X 250.3936, Y 44.2089, Z -6.3333, A 0.000, B 0.000, C 0.000 }
gfCNCPoint5[1074] = {X 250.3936, Y 45.0000, Z -6.3333, A 0.000, B 0.000, C 0.000 }
gfCNCPoint5[1075] = {X 250.2933, Y 45.8901, Z -6.3333, A 0.000, B 0.000, C 0.000 }
gfCNCPoint5[1076] = {X 249.9974, Y 46.7355, Z -6.3333, A 0.000, B 0.000, C 0.000 }
gfCNCPoint5[1077] = {X 249.5209, Y 47.4940, Z -6.3333, A 0.000, B 0.000, C 0.000 }
gfCNCPoint5[1078] = {X 248.8875, Y 48.1273, Z -6.3333, A 0.000, B 0.000, C 0.000 }
gfCNCPoint5[1079] = {X 248.1291, Y 48.6039, Z -6.3333, A 0.000, B 0.000, C 0.000 }
gfCNCPoint5[1080] = {X 247.2836, Y 48.8997, Z -6.3333, A 0.000, B 0.000, C 0.000 }
gfCNCPoint5[1081] = {X 246.3936, Y 49.0000, Z -6.3333, A 0.000, B 0.000, C 0.000 }
gfCNCPoint5[1082] = {X 239.8075, Y 49.0000, Z -6.3333, A 0.000, B 0.000, C 0.000 }
gfCNCPoint5[1083] = {X 238.9174, Y 48.8997, Z -6.3333, A 0.000, B 0.000, C 0.000 }
gfCNCPoint5[1084] = {X 238.0720, Y 48.6039, Z -6.3333, A 0.000, B 0.000, C 0.000 }
gfCNCPoint5[1085] = {X 237.3135, Y 48.1273, Z -6.3333, A 0.000, B 0.000, C 0.000 }
gfCNCPoint5[1086] = {X 236.6802, Y 47.4940, Z -6.3333, A 0.000, B 0.000, C 0.000 }
gfCNCPoint5[1087] = {X 236.2036, Y 46.7355, Z -6.3333, A 0.000, B 0.000, C 0.000 }
gfCNCPoint5[1088] = {X 235.9078, Y 45.8901, Z -6.3333, A 0.000, B 0.000, C 0.000 }
gfCNCPoint5[1089] = {X 235.8075, Y 45.0000, Z -6.3333, A 0.000, B 0.000, C 0.000 }
gfCNCPoint5[1090] = {X 235.8079, Y 44.1538, Z -6.3333, A 0.000, B 0.000, C 0.000 }
gfCNCPoint5[1091] = {X 235.9027, Y 43.3414, Z -6.3333, A 0.000, B 0.000, C 0.000 }
gfCNCPoint5[1092] = {X 236.1607, Y 42.5654, Z -6.3333, A 0.000, B 0.000, C 0.000 }
gfCNCPoint5[1093] = {X 236.5712, Y 41.8580, Z -6.3333, A 0.000, B 0.000, C 0.000 }
gfCNCPoint5[1094] = {X 237.1169, Y 41.2489, Z -6.3333, A 0.000, B 0.000, C 0.000 }
gfCNCPoint5[1095] = {X 237.7752, Y 40.7635, Z -6.3333, A 0.000, B 0.000, C 0.000 }
gfCNCPoint5[1096] = {X 238.5184, Y 40.4222, Z -6.3333, A 0.000, B 0.000, C 0.000 }
gfCNCPoint5[1097] = {X 242.7044, Y 32.2287, Z -6.3333, A 0.000, B 0.000, C 0.000 }
gfCNCPoint5[1098] = {X 241.5061, Y 31.4663, Z -6.3333, A 0.000, B 0.000, C 0.000 }
gfCNCPoint5[1099] = {X 240.4161, Y 30.5558, Z -6.3333, A 0.000, B 0.000, C 0.000 }
gfCNCPoint5[1100] = {X 239.4524, Y 29.5126, Z -6.3333, A 0.000, B 0.000, C 0.000 }
gfCNCPoint5[1101] = {X 238.6312, Y 28.3538, Z -6.3333, A 0.000, B 0.000, C 0.000 }
gfCNCPoint5[1102] = {X 237.9661, Y 27.0990, Z -6.3333, A 0.000, B 0.000, C 0.000 }
gfCNCPoint5[1103] = {X 237.4682, Y 25.7689, Z -6.3333, A 0.000, B 0.000, C 0.000 }
gfCNCPoint5[1104] = {X 237.0566, Y 23.9929, Z -6.3333, A 0.000, B 0.000, C 0.000 }
gfCNCPoint5[1105] = {X 236.8470, Y 22.1820, Z -6.3333, A 0.000, B 0.000, C 0.000 }
gfCNCPoint5[1106] = {X 236.8419, Y 20.3590, Z -6.3333, A 0.000, B 0.000, C 0.000 }
gfCNCPoint5[1107] = {X 237.0415, Y 18.5469, Z -6.3333, A 0.000, B 0.000, C 0.000 }
gfCNCPoint5[1108] = {X 237.4432, Y 16.7687, Z -6.3333, A 0.000, B 0.000, C 0.000 }
gfCNCPoint5[1109] = {X 237.9984, Y 15.2352, Z -6.3333, A 0.000, B 0.000, C 0.000 }
gfCNCPoint5[1110] = {X 238.7643, Y 13.7954, Z -6.3333, A 0.000, B 0.000, C 0.000 }
gfCNCPoint5[1111] = {X 239.7258, Y 12.4780, Z -6.3333, A 0.000, B 0.000, C 0.000 }
gfCNCPoint5[1112] = {X 240.8635, Y 11.3095, Z -6.3333, A 0.000, B 0.000, C 0.000 }
gfCNCPoint5[1113] = {X 242.1547, Y 10.3132, Z -6.3333, A 0.000, B 0.000, C 0.000 }
gfCNCPoint5[1114] = {X 243.5736, Y 9.5091, Z -6.3333, A 0.000, B 0.000, C 0.000 }
gfCNCPoint5[1115] = {X 245.0917, Y 8.9131, Z -6.3333, A 0.000, B 0.000, C 0.000 }
gfCNCPoint5[1116] = {X 246.6787, Y 8.5374, Z -6.3333, A 0.000, B 0.000, C 0.000 }
gfCNCPoint5[1117] = {X 248.7483, Y 8.2694, Z -6.3333, A 0.000, B 0.000, C 0.000 }
gfCNCPoint5[1118] = {X 250.8336, Y 8.1899, Z -6.3333, A 0.000, B 0.000, C 0.000 }
gfCNCPoint5[1119] = {X 266.7608, Y 8.1899, Z -6.3333, A 0.000, B 0.000, C 0.000 }
gfCNCPoint5[1120] = {X 267.6453, Y 8.2962, Z -6.3333, A 0.000, B 0.000, C 0.000 }
gfCNCPoint5[1121] = {X 268.4845, Y 8.5955, Z -6.3333, A 0.000, B 0.000, C 0.000 }
gfCNCPoint5[1122] = {X 269.2366, Y 9.0730, Z -6.3333, A 0.000, B 0.000, C 0.000 }
gfCNCPoint5[1123] = {X 269.8645, Y 9.7051, Z -6.3333, A 0.000, B 0.000, C 0.000 }
gfCNCPoint5[1124] = {X 270.3370, Y 10.4605, Z -6.3333, A 0.000, B 0.000, C 0.000 }
gfCNCPoint5[1125] = {X 270.6307, Y 11.3016, Z -6.3333, A 0.000, B 0.000, C 0.000 }
gfCNCPoint5[1126] = {X 270.7310, Y 12.1869, Z -6.3333, A 0.000, B 0.000, C 0.000 }
gfCNCPoint5[1127] = {X 270.7308, Y 13.0192, Z -6.3333, A 0.000, B 0.000, C 0.000 }
gfCNCPoint5[1128] = {X 270.6223, Y 13.9045, Z -6.3333, A 0.000, B 0.000, C 0.000 }
gfCNCPoint5[1129] = {X 270.3202, Y 14.7437, Z -6.3333, A 0.000, B 0.000, C 0.000 }
gfCNCPoint5[1130] = {X 269.8397, Y 15.4952, Z -6.3333, A 0.000, B 0.000, C 0.000 }
gfCNCPoint5[1131] = {X 269.2046, Y 16.1215, Z -6.3333, A 0.000, B 0.000, C 0.000 }
gfCNCPoint5[1132] = {X 269.2045, Y 28.5935, Z -6.3333, A 0.000, B 0.000, C 0.000 }
gfCNCPoint5[1133] = {X 273.2845, Y 28.5936, Z -6.3333, A 0.000, B 0.000, C 0.000 }
gfCNCPoint5[1134] = {X 273.2845, Y 28.5936, Z -3.3333, A 0.000, B 0.000, C 0.000 }
gfCNCPoint5[1135] = {X 273.2845, Y 28.5936, Z 11.0000, A 0.000, B 0.000, C 0.000 }
gfCNCPoint5[1136] = {X 277.7445, Y 28.5921, Z 11.0000, A 0.000, B 0.000, C 0.000 }
gfCNCPoint5[1137] = {X 277.7445, Y 28.5921, Z -3.3333, A 0.000, B 0.000, C 0.000 }
gfCNCPoint5[1138] = {X 277.7445, Y 28.5921, Z -6.3333, A 0.000, B 0.000, C 0.000 }
gfCNCPoint5[1139] = {X 281.8245, Y 28.5920, Z -6.3333, A 0.000, B 0.000, C 0.000 }
gfCNCPoint5[1140] = {X 281.8243, Y 16.2734, Z -6.3333, A 0.000, B 0.000, C 0.000 }
gfCNCPoint5[1141] = {X 281.1861, Y 15.6023, Z -6.3333, A 0.000, B 0.000, C 0.000 }
gfCNCPoint5[1142] = {X 280.7057, Y 14.8107, Z -6.3333, A 0.000, B 0.000, C 0.000 }
gfCNCPoint5[1143] = {X 280.4050, Y 13.9348, Z -6.3333, A 0.000, B 0.000, C 0.000 }
gfCNCPoint5[1144] = {X 280.2978, Y 13.0150, Z -6.3333, A 0.000, B 0.000, C 0.000 }
gfCNCPoint5[1145] = {X 280.2977, Y 12.1868, Z -6.3333, A 0.000, B 0.000, C 0.000 }
gfCNCPoint5[1146] = {X 280.4060, Y 11.2255, Z -6.3333, A 0.000, B 0.000, C 0.000 }
gfCNCPoint5[1147] = {X 280.7255, Y 10.3124, Z -6.3333, A 0.000, B 0.000, C 0.000 }
gfCNCPoint5[1148] = {X 281.2402, Y 9.4933, Z -6.3333, A 0.000, B 0.000, C 0.000 }
gfCNCPoint5[1149] = {X 281.9242, Y 8.8093, Z -6.3333, A 0.000, B 0.000, C 0.000 }
gfCNCPoint5[1150] = {X 282.7433, Y 8.2946, Z -6.3333, A 0.000, B 0.000, C 0.000 }
gfCNCPoint5[1151] = {X 283.6564, Y 7.9751, Z -6.3333, A 0.000, B 0.000, C 0.000 }
gfCNCPoint5[1152] = {X 284.6177, Y 7.8668, Z -6.3333, A 0.000, B 0.000, C 0.000 }
gfCNCPoint5[1153] = {X 291.0611, Y 7.8668, Z -6.3333, A 0.000, B 0.000, C 0.000 }
gfCNCPoint5[1154] = {X 292.0224, Y 7.9751, Z -6.3333, A 0.000, B 0.000, C 0.000 }
gfCNCPoint5[1155] = {X 292.9355, Y 8.2946, Z -6.3333, A 0.000, B 0.000, C 0.000 }
gfCNCPoint5[1156] = {X 293.7546, Y 8.8093, Z -6.3333, A 0.000, B 0.000, C 0.000 }
gfCNCPoint5[1157] = {X 294.4386, Y 9.4933, Z -6.3333, A 0.000, B 0.000, C 0.000 }
gfCNCPoint5[1158] = {X 294.9533, Y 10.3124, Z -6.3333, A 0.000, B 0.000, C 0.000 }
gfCNCPoint5[1159] = {X 295.2728, Y 11.2255, Z -6.3333, A 0.000, B 0.000, C 0.000 }
gfCNCPoint5[1160] = {X 295.3811, Y 12.1868, Z -6.3333, A 0.000, B 0.000, C 0.000 }
gfCNCPoint5[1161] = {X 295.3811, Y 12.9782, Z -6.3333, A 0.000, B 0.000, C 0.000 }
gfCNCPoint5[1162] = {X 295.2798, Y 13.9079, Z -6.3333, A 0.000, B 0.000, C 0.000 }
gfCNCPoint5[1163] = {X 294.9807, Y 14.7940, Z -6.3333, A 0.000, B 0.000, C 0.000 }
gfCNCPoint5[1164] = {X 294.4980, Y 15.5949, Z -6.3333, A 0.000, B 0.000, C 0.000 }
gfCNCPoint5[1165] = {X 293.8542, Y 16.2733, Z -6.3333, A 0.000, B 0.000, C 0.000 }
gfCNCPoint5[1166] = {X 293.8552, Y 22.1965, Z -6.3333, A 0.000, B 0.000, C 0.000 }
gfCNCPoint5[1167] = {X 302.7587, Y 22.1965, Z -6.3333, A 0.000, B 0.000, C 0.000 }
gfCNCPoint5[1168] = {X 302.7637, Y 16.2775, Z -6.3333, A 0.000, B 0.000, C 0.000 }
gfCNCPoint5[1169] = {X 302.1238, Y 15.6064, Z -6.3333, A 0.000, B 0.000, C 0.000 }
gfCNCPoint5[1170] = {X 301.6419, Y 14.8142, Z -6.3333, A 0.000, B 0.000, C 0.000 }
gfCNCPoint5[1171] = {X 301.3402, Y 13.9375, Z -6.3333, A 0.000, B 0.000, C 0.000 }
gfCNCPoint5[1172] = {X 301.2324, Y 13.0165, Z -6.3333, A 0.000, B 0.000, C 0.000 }
gfCNCPoint5[1173] = {X 301.2323, Y 12.1868, Z -6.3333, A 0.000, B 0.000, C 0.000 }
gfCNCPoint5[1174] = {X 301.3406, Y 11.2255, Z -6.3333, A 0.000, B 0.000, C 0.000 }
gfCNCPoint5[1175] = {X 301.6601, Y 10.3124, Z -6.3333, A 0.000, B 0.000, C 0.000 }
gfCNCPoint5[1176] = {X 302.1747, Y 9.4933, Z -6.3333, A 0.000, B 0.000, C 0.000 }
gfCNCPoint5[1177] = {X 302.8588, Y 8.8093, Z -6.3333, A 0.000, B 0.000, C 0.000 }
gfCNCPoint5[1178] = {X 303.6779, Y 8.2946, Z -6.3333, A 0.000, B 0.000, C 0.000 }
gfCNCPoint5[1179] = {X 304.5910, Y 7.9751, Z -6.3333, A 0.000, B 0.000, C 0.000 }
gfCNCPoint5[1180] = {X 305.5523, Y 7.8668, Z -6.3333, A 0.000, B 0.000, C 0.000 }
gfCNCPoint5[1181] = {X 311.9957, Y 7.8668, Z -6.3333, A 0.000, B 0.000, C 0.000 }
gfCNCPoint5[1182] = {X 312.9570, Y 7.9751, Z -6.3333, A 0.000, B 0.000, C 0.000 }
gfCNCPoint5[1183] = {X 313.8701, Y 8.2946, Z -6.3333, A 0.000, B 0.000, C 0.000 }
gfCNCPoint5[1184] = {X 314.6892, Y 8.8093, Z -6.3333, A 0.000, B 0.000, C 0.000 }
gfCNCPoint5[1185] = {X 315.3732, Y 9.4933, Z -6.3333, A 0.000, B 0.000, C 0.000 }
gfCNCPoint5[1186] = {X 315.8879, Y 10.3124, Z -6.3333, A 0.000, B 0.000, C 0.000 }
gfCNCPoint5[1187] = {X 316.2074, Y 11.2255, Z -6.3333, A 0.000, B 0.000, C 0.000 }
gfCNCPoint5[1188] = {X 316.3157, Y 12.1868, Z -6.3333, A 0.000, B 0.000, C 0.000 }
gfCNCPoint5[1189] = {X 316.3157, Y 12.9782, Z -6.3333, A 0.000, B 0.000, C 0.000 }
gfCNCPoint5[1190] = {X 316.2145, Y 13.9077, Z -6.3333, A 0.000, B 0.000, C 0.000 }
gfCNCPoint5[1191] = {X 315.9156, Y 14.7937, Z -6.3333, A 0.000, B 0.000, C 0.000 }
gfCNCPoint5[1192] = {X 315.4331, Y 15.5947, Z -6.3333, A 0.000, B 0.000, C 0.000 }
gfCNCPoint5[1193] = {X 314.7895, Y 16.2730, Z -6.3333, A 0.000, B 0.000, C 0.000 }
gfCNCPoint5[1194] = {X 314.7887, Y 40.9131, Z -6.3333, A 0.000, B 0.000, C 0.000 }
gfCNCPoint5[1195] = {X 315.4269, Y 41.5841, Z -6.3333, A 0.000, B 0.000, C 0.000 }
gfCNCPoint5[1196] = {X 315.9075, Y 42.3757, Z -6.3333, A 0.000, B 0.000, C 0.000 }
gfCNCPoint5[1197] = {X 316.2083, Y 43.2515, Z -6.3333, A 0.000, B 0.000, C 0.000 }
gfCNCPoint5[1198] = {X 316.3156, Y 44.1713, Z -6.3333, A 0.000, B 0.000, C 0.000 }
gfCNCPoint5[1199] = {X 316.3157, Y 45.0000, Z -6.3333, A 0.000, B 0.000, C 0.000 }
gfCNCPoint5[1200] = {X 316.2074, Y 45.9613, Z -6.3333, A 0.000, B 0.000, C 0.000 }
gfCNCPoint5[1201] = {X 315.8879, Y 46.8744, Z -6.3333, A 0.000, B 0.000, C 0.000 }
gfCNCPoint5[1202] = {X 315.3732, Y 47.6935, Z -6.3333, A 0.000, B 0.000, C 0.000 }
gfCNCPoint5[1203] = {X 314.6892, Y 48.3775, Z -6.3333, A 0.000, B 0.000, C 0.000 }
gfCNCPoint5[1204] = {X 313.8701, Y 48.8922, Z -6.3333, A 0.000, B 0.000, C 0.000 }
gfCNCPoint5[1205] = {X 312.9570, Y 49.2117, Z -6.3333, A 0.000, B 0.000, C 0.000 }
gfCNCPoint5[1206] = {X 311.9957, Y 49.3200, Z -6.3333, A 0.000, B 0.000, C 0.000 }
gfCNCPoint5[1207] = {X 305.5523, Y 49.3200, Z -6.3333, A 0.000, B 0.000, C 0.000 }
gfCNCPoint5[1208] = {X 304.5958, Y 49.2128, Z -6.3333, A 0.000, B 0.000, C 0.000 }
gfCNCPoint5[1209] = {X 303.6868, Y 48.8965, Z -6.3333, A 0.000, B 0.000, C 0.000 }
gfCNCPoint5[1210] = {X 302.8704, Y 48.3868, Z -6.3333, A 0.000, B 0.000, C 0.000 }
gfCNCPoint5[1211] = {X 302.1872, Y 47.7090, Z -6.3333, A 0.000, B 0.000, C 0.000 }
gfCNCPoint5[1212] = {X 301.6709, Y 46.8967, Z -6.3333, A 0.000, B 0.000, C 0.000 }
gfCNCPoint5[1213] = {X 301.3473, Y 45.9903, Z -6.3333, A 0.000, B 0.000, C 0.000 }
gfCNCPoint5[1214] = {X 301.2324, Y 45.0348, Z -6.3333, A 0.000, B 0.000, C 0.000 }
gfCNCPoint5[1215] = {X 301.2323, Y 44.2013, Z -6.3333, A 0.000, B 0.000, C 0.000 }
gfCNCPoint5[1216] = {X 301.3496, Y 43.2652, Z -6.3333, A 0.000, B 0.000, C 0.000 }
gfCNCPoint5[1217] = {X 301.6526, Y 42.3718, Z -6.3333, A 0.000, B 0.000, C 0.000 }
gfCNCPoint5[1218] = {X 302.1289, Y 41.5574, Z -6.3333, A 0.000, B 0.000, C 0.000 }
gfCNCPoint5[1219] = {X 302.7591, Y 40.8553, Z -6.3333, A 0.000, B 0.000, C 0.000 }
